LIN {X 0,Y 246.822,Z 659.839,A -85,B 0,C 180,E1 -20933.784,E2 -20933.784} C_VEL
LIN {X 0,Y 240.149,Z 668.993,A -85,B 0,C 180,E1 -20935.712,E2 -20935.712} C_VEL
LIN {X 0,Y 234.092,Z 676.593,A -85,B 0,C 180,E1 -20937.798,E2 -20937.798} C_VEL
LIN {X 0,Y 227.642,Z 683.866,A -85,B 0,C 180,E1 -20940.398,E2 -20940.398} C_VEL
LIN {X 0,Y 222.706,Z 688.862,A -85,B 0,C 180,E1 -20942.769,E2 -20942.769} C_VEL
LIN {X 0,Y 218.214,Z 692.902,A -85,B 0,C 180,E1 -20945.248,E2 -20945.248} C_VEL
LIN {X 0,Y 215.578,Z 695.042,A -85,B 0,C 180,E1 -20946.97,E2 -20946.97} C_VEL
LIN {X 0,Y 211.246,Z 698.163,A -85,B 0,C 180,E1 -20950.568,E2 -20950.568} C_VEL
LIN {X 0,Y 208.028,Z 699.817,A -85,B 0,C 180,E1 -20954.32,E2 -20954.32} C_VEL
LIN {X 0,Y 205.977,Z 699.948,A -85,B 0,C 180,E1 -20958.187,E2 -20958.187} C_VEL
LIN {X 0,Y 204.89,Z 698.61,A -85,B 0,C 180,E1 -20962.114,E2 -20962.114} C_VEL
LIN {X 0,Y 204.811,Z 698.606,A -85,B 0,C 180,E1 -20962.607,E2 -20962.607} C_VEL
LIN {X 0,Y 204.425,Z 700.65,A -85,B 0,C 180,E1 -20966.057,E2 -20966.057} C_VEL
LIN {X 0,Y 204.43,Z 701.266,A -85,B 0,C 180,E1 -20968.03,E2 -20968.03} C_VEL
LIN {X 0,Y 204.516,Z 701.484,A -85,B 0,C 180,E1 -20970,E2 -20970} C_VEL
LIN {X 0,Y 204.399,Z 701.253,A -85,B 0,C 180,E1 -20971.97,E2 -20971.97} C_VEL
LIN {X 0,Y 204.384,Z 700.488,A -85,B 0,C 180,E1 -20974.287,E2 -20974.287} C_VEL
LIN {X 0,Y 204.663,Z 698.173,A -85,B 0,C 180,E1 -20977.895,E2 -20977.895} C_VEL
LIN {X 0,Y 205.307,Z 695.187,A -85,B 0,C 180,E1 -20980.852,E2 -20980.852} C_VEL
LIN {X 0,Y 206.295,Z 691.137,A -85,B 0,C 180,E1 -20983.797,E2 -20983.797} C_VEL
LIN {X 0,Y 208.254,Z 684.908,A -85,B 0,C 180,E1 -20987.175,E2 -20987.175} C_VEL
LIN {X 0,Y 210.401,Z 678.115,A -85,B 0,C 180,E1 -20990.022,E2 -20990.022} C_VEL
LIN {X 0,Y 212.491,Z 671.31,A -85,B 0,C 180,E1 -20992.394,E2 -20992.394} C_VEL
LIN {X 0,Y 217.207,Z 666.561,A -85,B 0,C 180,E1 -20995.901,E2 -20995.901} C_VEL
LIN {X 0,Y 221.61,Z 661.924,A -85,B 0,C 180,E1 -20998.405,E2 -20998.405} C_VEL
LIN {X 0,Y 227.57,Z 655.288,A -85,B 0,C 180,E1 -21001.151,E2 -21001.151} C_VEL
LIN {X 0,Y 234.374,Z 647.105,A -85,B 0,C 180,E1 -21003.693,E2 -21003.693} C_VEL
LIN {X 0,Y 241.865,Z 637.223,A -85,B 0,C 180,E1 -21006.045,E2 -21006.045} C_VEL
LIN {X 0,Y 249.165,Z 626.646,A -85,B 0,C 180,E1 -21007.894,E2 -21007.894} C_VEL
LIN {X 0,Y 255.952,Z 615.572,A -85,B 0,C 180,E1 -21009.418,E2 -21009.418} C_VEL
LIN {X 0,Y 262.663,Z 603.149,A -85,B 0,C 180,E1 -21010.708,E2 -21010.708} C_VEL
LIN {X 0,Y 269.007,Z 589.494,A -85,B 0,C 180,E1 -21011.775,E2 -21011.775} C_VEL
LIN {X 0,Y 275.128,Z 573.285,A -85,B 0,C 180,E1 -21012.729,E2 -21012.729} C_VEL
LIN {X 0,Y 279.953,Z 556.394,A -85,B 0,C 180,E1 -21013.539,E2 -21013.539} C_VEL
LIN {X 0,Y 281.282,Z 550.85,A -85,B 0,C 180,E1 -21013.828,E2 -21013.828} C_VEL
LIN {X 0,Y 282.041,Z 547.448,A -85,B 0,C 180,E1 -21014.196,E2 -21014.196} C_VEL
LIN {X 0,Y 282.381,Z 544.653,A -85,B 0,C 180,E1 -21016.2,E2 -21016.2} C_VEL
LIN {X 0,Y 282.787,Z 543.852,A -85,B 0,C 180,E1 -21017.546,E2 -21017.546} C_VEL
LIN {X 0,Y 277.691,Z 563.088,A -85,B 0,C 180,E1 -21018.619,E2 -21018.619} C_VEL
LIN {X 0,Y 272.938,Z 576.661,A -85,B 0,C 180,E1 -21019.687,E2 -21019.687} C_VEL
LIN {X 0,Y 267.626,Z 588.882,A -85,B 0,C 180,E1 -21020.931,E2 -21020.931} C_VEL
LIN {X 0,Y 261.853,Z 600.028,A -85,B 0,C 180,E1 -21022.367,E2 -21022.367} C_VEL
LIN {X 0,Y 255.179,Z 610.907,A -85,B 0,C 180,E1 -21024.179,E2 -21024.179} C_VEL
LIN {X 0,Y 248.845,Z 619.829,A -85,B 0,C 180,E1 -21026.097,E2 -21026.097} C_VEL
LIN {X 0,Y 242.801,Z 627.197,A -85,B 0,C 180,E1 -21028.112,E2 -21028.112} C_VEL
LIN {X 0,Y 236.398,Z 634.071,A -85,B 0,C 180,E1 -21030.624,E2 -21030.624} C_VEL
LIN {X 0,Y 231.215,Z 638.794,A -85,B 0,C 180,E1 -21032.875,E2 -21032.875} C_VEL
LIN {X 0,Y 225.025,Z 643.457,A -85,B 0,C 180,E1 -21036.045,E2 -21036.045} C_VEL
LIN {X 0,Y 222.181,Z 645.2,A -85,B 0,C 180,E1 -21037.692,E2 -21037.692} C_VEL
LIN {X 0,Y 219.568,Z 646.531,A -85,B 0,C 180,E1 -21039.385,E2 -21039.385} C_VEL
LIN {X 0,Y 217.066,Z 647.461,A -85,B 0,C 180,E1 -21041.109,E2 -21041.109} C_VEL
LIN {X 0,Y 212.867,Z 648.156,A -85,B 0,C 180,E1 -21044.685,E2 -21044.685} C_VEL
LIN {X 0,Y 211.13,Z 647.932,A -85,B 0,C 180,E1 -21046.526,E2 -21046.526} C_VEL
LIN {X 0,Y 208.468,Z 646.274,A -85,B 0,C 180,E1 -21050.296,E2 -21050.296} C_VEL
LIN {X 0,Y 206.567,Z 643.065,A -85,B 0,C 180,E1 -21054.142,E2 -21054.142} C_VEL
LIN {X 0,Y 205.609,Z 639.573,A -85,B 0,C 180,E1 -21057.061,E2 -21057.061} C_VEL
LIN {X 0,Y 205.18,Z 635.056,A -85,B 0,C 180,E1 -21060,E2 -21060} C_VEL
LIN {X 0,Y 205.28,Z 628.361,A -85,B 0,C 180,E1 -21063.435,E2 -21063.435} C_VEL
LIN {X 0,Y 205.557,Z 622.501,A -85,B 0,C 180,E1 -21065.887,E2 -21065.887} C_VEL
LIN {X 0,Y 205.965,Z 613.792,A -85,B 0,C 180,E1 -21068.89,E2 -21068.89} C_VEL
LIN {X 0,Y 206.717,Z 603.469,A -85,B 0,C 180,E1 -21071.77,E2 -21071.77} C_VEL
LIN {X 0,Y 207.701,Z 591.458,A -85,B 0,C 180,E1 -21074.451,E2 -21074.451} C_VEL
LIN {X 0,Y 208.737,Z 579.31,A -85,B 0,C 180,E1 -21076.63,E2 -21076.63} C_VEL
LIN {X 0,Y 209.825,Z 565.811,A -85,B 0,C 180,E1 -21078.554,E2 -21078.554} C_VEL
LIN {X 0,Y 210.638,Z 551.375,A -85,B 0,C 180,E1 -21080.114,E2 -21080.114} C_VEL
LIN {X 0,Y 211.452,Z 537.597,A -85,B 0,C 180,E1 -21081.197,E2 -21081.197} C_VEL
LIN {X 0,Y 214.083,Z 473.822,A -85,B 0,C 180,E1 -21084.869,E2 -21084.869} C_VEL
LIN {X 0,Y 207.846,Z 451.881,A -85,B 0,C 180,E1 -21086.423,E2 -21086.423} C_VEL
LIN {X 0,Y 206.822,Z 447.715,A -85,B 0,C 180,E1 -21086.741,E2 -21086.741} C_VEL
LIN {X 0,Y 206.719,Z 447.71,A -85,B 0,C 180,E1 -21091.794,E2 -21091.794} C_VEL
LIN {X 0,Y 206.701,Z 447.709,A -85,B 0,C 180,E1 -21095.311,E2 -21095.311} C_VEL
LIN {X 0,Y 206.657,Z 447.832,A -85,B 0,C 180,E1 -21099.431,E2 -21099.431} C_VEL
LIN {X 0,Y 207.094,Z 449.45,A -85,B 0,C 180,E1 -21100.15,E2 -21100.15} C_VEL
LIN {X 0,Y 208.097,Z 451.279,A -85,B 0,C 180,E1 -21101.101,E2 -21101.101} C_VEL
LIN {X 0,Y 211.34,Z 459.761,A -85,B 0,C 180,E1 -21104.839,E2 -21104.839} C_VEL
LIN {X 0,Y 214.271,Z 468.248,A -85,B 0,C 180,E1 -21108.223,E2 -21108.223} C_VEL
LIN {X 0,Y 216.652,Z 475.96,A -85,B 0,C 180,E1 -21110.943,E2 -21110.943} C_VEL
LIN {X 0,Y 222.997,Z 488.678,A -85,B 0,C 180,E1 -21112.765,E2 -21112.765} C_VEL
LIN {X 0,Y 228.7,Z 501.914,A -85,B 0,C 180,E1 -21114.352,E2 -21114.352} C_VEL
LIN {X 0,Y 231.099,Z 518.723,A -85,B 0,C 180,E1 -21115.406,E2 -21115.406} C_VEL
LIN {X 0,Y 228.053,Z 586.183,A -85,B 0,C 180,E1 -21117.429,E2 -21117.429} C_VEL
LIN {X 0,Y 226.882,Z 599.328,A -85,B 0,C 180,E1 -21118.093,E2 -21118.093} C_VEL
LIN {X 0,Y 225.302,Z 611.278,A -85,B 0,C 180,E1 -21119.023,E2 -21119.023} C_VEL
LIN {X 0,Y 223.274,Z 622.987,A -85,B 0,C 180,E1 -21120.28,E2 -21120.28} C_VEL
LIN {X 0,Y 220.717,Z 635.03,A -85,B 0,C 180,E1 -21121.987,E2 -21121.987} C_VEL
LIN {X 0,Y 218.056,Z 645.622,A -85,B 0,C 180,E1 -21123.951,E2 -21123.951} C_VEL
LIN {X 0,Y 215.52,Z 654.872,A -85,B 0,C 180,E1 -21126.12,E2 -21126.12} C_VEL
LIN {X 0,Y 212.898,Z 663.681,A -85,B 0,C 180,E1 -21128.708,E2 -21128.708} C_VEL
LIN {X 0,Y 210.376,Z 671.148,A -85,B 0,C 180,E1 -21131.496,E2 -21131.496} C_VEL
LIN {X 0,Y 208.434,Z 677.133,A -85,B 0,C 180,E1 -21134.351,E2 -21134.351} C_VEL
LIN {X 0,Y 206.83,Z 681.865,A -85,B 0,C 180,E1 -21137.24,E2 -21137.24} C_VEL
LIN {X 0,Y 205.714,Z 685.481,A -85,B 0,C 180,E1 -21140.164,E2 -21140.164} C_VEL
LIN {X 0,Y 205.197,Z 687.34,A -85,B 0,C 180,E1 -21142.126,E2 -21142.126} C_VEL
LIN {X 0,Y 204.763,Z 688.973,A -85,B 0,C 180,E1 -21144.479,E2 -21144.479} C_VEL
LIN {X 0,Y 204.472,Z 690.36,A -85,B 0,C 180,E1 -21148.03,E2 -21148.03} C_VEL
LIN {X 0,Y 204.474,Z 690.59,A -85,B 0,C 180,E1 -21150,E2 -21150} C_VEL
LIN {X 0,Y 204.471,Z 690.394,A -85,B 0,C 180,E1 -21151.97,E2 -21151.97} C_VEL
LIN {X 0,Y 204.823,Z 688.834,A -85,B 0,C 180,E1 -21155.908,E2 -21155.908} C_VEL
LIN {X 0,Y 205.193,Z 687.462,A -85,B 0,C 180,E1 -21157.874,E2 -21157.874} C_VEL
LIN {X 0,Y 206.024,Z 684.579,A -85,B 0,C 180,E1 -21160.814,E2 -21160.814} C_VEL
LIN {X 0,Y 207.272,Z 680.658,A -85,B 0,C 180,E1 -21163.73,E2 -21163.73} C_VEL
LIN {X 0,Y 208.976,Z 675.573,A -85,B 0,C 180,E1 -21166.61,E2 -21166.61} C_VEL
LIN {X 0,Y 211.126,Z 669.161,A -85,B 0,C 180,E1 -21169.444,E2 -21169.444} C_VEL
LIN {X 0,Y 213.778,Z 661.188,A -85,B 0,C 180,E1 -21172.214,E2 -21172.214} C_VEL
LIN {X 0,Y 216.312,Z 652.44,A -85,B 0,C 180,E1 -21174.642,E2 -21174.642} C_VEL
LIN {X 0,Y 218.833,Z 642.979,A -85,B 0,C 180,E1 -21176.719,E2 -21176.719} C_VEL
LIN {X 0,Y 221.597,Z 631.665,A -85,B 0,C 180,E1 -21178.665,E2 -21178.665} C_VEL
LIN {X 0,Y 223.833,Z 620.502,A -85,B 0,C 180,E1 -21180.157,E2 -21180.157} C_VEL
LIN {X 0,Y 225.952,Z 607.822,A -85,B 0,C 180,E1 -21181.399,E2 -21181.399} C_VEL
LIN {X 0,Y 227.283,Z 596.137,A -85,B 0,C 180,E1 -21182.236,E2 -21182.236} C_VEL
LIN {X 0,Y 228.293,Z 583.8,A -85,B 0,C 180,E1 -21182.794,E2 -21182.794} C_VEL
LIN {X 0,Y 231.175,Z 518.266,A -85,B 0,C 180,E1 -21184.746,E2 -21184.746} C_VEL
LIN {X 0,Y 228.56,Z 501.373,A -85,B 0,C 180,E1 -21185.844,E2 -21185.844} C_VEL
LIN {X 0,Y 222.629,Z 487.777,A -85,B 0,C 180,E1 -21187.498,E2 -21187.498} C_VEL
LIN {X 0,Y 216.547,Z 475.617,A -85,B 0,C 180,E1 -21189.3,E2 -21189.3} C_VEL
LIN {X 0,Y 213.479,Z 465.768,A -85,B 0,C 180,E1 -21192.903,E2 -21192.903} C_VEL
LIN {X 0,Y 210.639,Z 457.862,A -85,B 0,C 180,E1 -21196.186,E2 -21196.186} C_VEL
LIN {X 0,Y 207.768,Z 450.735,A -85,B 0,C 180,E1 -21199.388,E2 -21199.388} C_VEL
LIN {X 0,Y 206.681,Z 447.744,A -85,B 0,C 180,E1 -21200.807,E2 -21200.807} C_VEL
LIN {X 0,Y 206.798,Z 447.743,A -85,B 0,C 180,E1 -21204.357,E2 -21204.357} C_VEL
LIN {X 0,Y 210.172,Z 463.929,A -85,B 0,C 180,E1 -21209.061,E2 -21209.061} C_VEL
LIN {X 0,Y 212.003,Z 472.76,A -85,B 0,C 180,E1 -21211.54,E2 -21211.54} C_VEL
LIN {X 0,Y 211.794,Z 476.671,A -85,B 0,C 180,E1 -21212.515,E2 -21212.515} C_VEL
LIN {X 0,Y 213.201,Z 497.323,A -85,B 0,C 180,E1 -21213.773,E2 -21213.773} C_VEL
LIN {X 0,Y 214.619,Z 511.272,A -85,B 0,C 180,E1 -21214.629,E2 -21214.629} C_VEL
LIN {X 0,Y 210.995,Z 588.15,A -85,B 0,C 180,E1 -21219.055,E2 -21219.055} C_VEL
LIN {X 0,Y 210.145,Z 602.588,A -85,B 0,C 180,E1 -21220.272,E2 -21220.272} C_VEL
LIN {X 0,Y 209.238,Z 614.678,A -85,B 0,C 180,E1 -21221.646,E2 -21221.646} C_VEL
LIN {X 0,Y 208.238,Z 627.949,A -85,B 0,C 180,E1 -21223.581,E2 -21223.581} C_VEL
LIN {X 0,Y 207.079,Z 640.895,A -85,B 0,C 180,E1 -21226.006,E2 -21226.006} C_VEL
LIN {X 0,Y 206.541,Z 646.882,A -85,B 0,C 180,E1 -21227.351,E2 -21227.351} C_VEL
LIN {X 0,Y 205.425,Z 651.21,A -85,B 0,C 180,E1 -21228.448,E2 -21228.448} C_VEL
LIN {X 0,Y 202.035,Z 657.624,A -85,B 0,C 180,E1 -21230.368,E2 -21230.368} C_VEL
LIN {X 0,Y 198.845,Z 663.489,A -85,B 0,C 180,E1 -21232.472,E2 -21232.472} C_VEL
LIN {X 0,Y 198.045,Z 667.005,A -85,B 0,C 180,E1 -21233.822,E2 -21233.822} C_VEL
LIN {X 0,Y 197.791,Z 674.226,A -85,B 0,C 180,E1 -21236.945,E2 -21236.945} C_VEL
LIN {X 0,Y 197.636,Z 679.846,A -85,B 0,C 180,E1 -21240,E2 -21240} C_VEL
LIN {X 0,Y 197.667,Z 684.221,A -85,B 0,C 180,E1 -21243.057,E2 -21243.057} C_VEL
LIN {X 0,Y 197.997,Z 687.774,A -85,B 0,C 180,E1 -21246.342,E2 -21246.342} C_VEL
LIN {X 0,Y 199.157,Z 690.616,A -85,B 0,C 180,E1 -21250.163,E2 -21250.163} C_VEL
LIN {X 0,Y 200.099,Z 691.561,A -85,B 0,C 180,E1 -21252.165,E2 -21252.165} C_VEL
LIN {X 0,Y 202.85,Z 692.291,A -85,B 0,C 180,E1 -21256.091,E2 -21256.091} C_VEL
LIN {X 0,Y 206.515,Z 691.591,A -85,B 0,C 180,E1 -21259.896,E2 -21259.896} C_VEL
LIN {X 0,Y 211.509,Z 689.338,A -85,B 0,C 180,E1 -21263.499,E2 -21263.499} C_VEL
LIN {X 0,Y 217.38,Z 685.573,A -85,B 0,C 180,E1 -21266.912,E2 -21266.912} C_VEL
LIN {X 0,Y 222.428,Z 681.658,A -85,B 0,C 180,E1 -21269.324,E2 -21269.324} C_VEL
LIN {X 0,Y 227.95,Z 676.712,A -85,B 0,C 180,E1 -21271.61,E2 -21271.61} C_VEL
LIN {X 0,Y 234.961,Z 669.564,A -85,B 0,C 180,E1 -21274.114,E2 -21274.114} C_VEL
LIN {X 0,Y 242.537,Z 660.638,A -85,B 0,C 180,E1 -21276.443,E2 -21276.443} C_VEL
LIN {X 0,Y 249.499,Z 651.211,A -85,B 0,C 180,E1 -21278.295,E2 -21278.295} C_VEL
LIN {X 0,Y 256.842,Z 639.775,A -85,B 0,C 180,E1 -21280.019,E2 -21280.019} C_VEL
LIN {X 0,Y 263.232,Z 628.029,A -85,B 0,C 180,E1 -21281.361,E2 -21281.361} C_VEL
LIN {X 0,Y 269.285,Z 614.812,A -85,B 0,C 180,E1 -21282.478,E2 -21282.478} C_VEL
LIN {X 0,Y 273.318,Z 604.09,A -85,B 0,C 180,E1 -21283.161,E2 -21283.161} C_VEL
LIN {X 0,Y 277.995,Z 588.116,A -85,B 0,C 180,E1 -21283.92,E2 -21283.92} C_VEL
LIN {X 0,Y 283.776,Z 566.322,A -85,B 0,C 180,E1 -21284.857,E2 -21284.857} C_VEL
LIN {X 0,Y 283.782,Z 566.28,A -85,B 0,C 180,E1 -21284.988,E2 -21284.988} C_VEL
LIN {X 0,Y 274.469,Z 600.667,A -85,B 0,C 180,E1 -21286.489,E2 -21286.489} C_VEL
LIN {X 0,Y 269.264,Z 615.152,A -85,B 0,C 180,E1 -21287.264,E2 -21287.264} C_VEL
LIN {X 0,Y 263.479,Z 628.141,A -85,B 0,C 180,E1 -21288.176,E2 -21288.176} C_VEL
LIN {X 0,Y 257.251,Z 639.905,A -85,B 0,C 180,E1 -21289.288,E2 -21289.288} C_VEL
LIN {X 0,Y 251.316,Z 649.663,A -85,B 0,C 180,E1 -21290.491,E2 -21290.491} C_VEL
LIN {X 0,Y 243.861,Z 660.474,A -85,B 0,C 180,E1 -21292.235,E2 -21292.235} C_VEL
LIN {X 0,Y 236.866,Z 669.428,A -85,B 0,C 180,E1 -21294.126,E2 -21294.126} C_VEL
LIN {X 0,Y 230.383,Z 676.825,A -85,B 0,C 180,E1 -21296.17,E2 -21296.17} C_VEL
LIN {X 0,Y 223.515,Z 683.927,A -85,B 0,C 180,E1 -21298.747,E2 -21298.747} C_VEL
LIN {X 0,Y 216.518,Z 690.243,A -85,B 0,C 180,E1 -21301.923,E2 -21301.923} C_VEL
LIN {X 0,Y 211.85,Z 693.85,A -85,B 0,C 180,E1 -21304.452,E2 -21304.452} C_VEL
LIN {X 0,Y 209.116,Z 695.783,A -85,B 0,C 180,E1 -21306.215,E2 -21306.215} C_VEL
LIN {X 0,Y 204.568,Z 698.452,A -85,B 0,C 180,E1 -21309.906,E2 -21309.906} C_VEL
LIN {X 0,Y 201.182,Z 699.686,A -85,B 0,C 180,E1 -21313.771,E2 -21313.771} C_VEL
LIN {X 0,Y 199.019,Z 699.489,A -85,B 0,C 180,E1 -21317.767,E2 -21317.767} C_VEL
LIN {X 0,Y 197.914,Z 697.929,A -85,B 0,C 180,E1 -21321.705,E2 -21321.705} C_VEL
LIN {X 0,Y 197.348,Z 700.363,A -85,B 0,C 180,E1 -21325.668,E2 -21325.668} C_VEL
LIN {X 0,Y 197.334,Z 701.077,A -85,B 0,C 180,E1 -21327.959,E2 -21327.959} C_VEL
LIN {X 0,Y 197.414,Z 701.295,A -85,B 0,C 180,E1 -21330,E2 -21330} C_VEL
LIN {X 0,Y 197.303,Z 701.064,A -85,B 0,C 180,E1 -21332.041,E2 -21332.041} C_VEL
LIN {X 0,Y 197.286,Z 700.44,A -85,B 0,C 180,E1 -21334.086,E2 -21334.086} C_VEL
LIN {X 0,Y 197.366,Z 699.423,A -85,B 0,C 180,E1 -21336.132,E2 -21336.132} C_VEL
LIN {X 0,Y 197.608,Z 697.982,A -85,B 0,C 180,E1 -21338.179,E2 -21338.179} C_VEL
LIN {X 0,Y 198.292,Z 694.996,A -85,B 0,C 180,E1 -21341.241,E2 -21341.241} C_VEL
LIN {X 0,Y 199.367,Z 690.947,A -85,B 0,C 180,E1 -21344.286,E2 -21344.286} C_VEL
LIN {X 0,Y 201.469,Z 684.719,A -85,B 0,C 180,E1 -21347.772,E2 -21347.772} C_VEL
LIN {X 0,Y 203.708,Z 678,A -85,B 0,C 180,E1 -21350.678,E2 -21350.678} C_VEL
LIN {X 0,Y 205.782,Z 671.436,A -85,B 0,C 180,E1 -21353.02,E2 -21353.02} C_VEL
LIN {X 0,Y 209.471,Z 668.21,A -85,B 0,C 180,E1 -21355.86,E2 -21355.86} C_VEL
LIN {X 0,Y 215.452,Z 662.758,A -85,B 0,C 180,E1 -21359.295,E2 -21359.295} C_VEL
LIN {X 0,Y 220.662,Z 657.61,A -85,B 0,C 180,E1 -21361.703,E2 -21361.703} C_VEL
LIN {X 0,Y 227.571,Z 650.286,A -85,B 0,C 180,E1 -21364.306,E2 -21364.306} C_VEL
LIN {X 0,Y 235.199,Z 641.371,A -85,B 0,C 180,E1 -21366.7,E2 -21366.7} C_VEL
LIN {X 0,Y 242.388,Z 632.189,A -85,B 0,C 180,E1 -21368.565,E2 -21368.565} C_VEL
LIN {X 0,Y 250.724,Z 620.207,A -85,B 0,C 180,E1 -21370.407,E2 -21370.407} C_VEL
LIN {X 0,Y 257.612,Z 609.046,A -85,B 0,C 180,E1 -21371.681,E2 -21371.681} C_VEL
LIN {X 0,Y 264.024,Z 597.055,A -85,B 0,C 180,E1 -21372.749,E2 -21372.749} C_VEL
LIN {X 0,Y 270.001,Z 584.082,A -85,B 0,C 180,E1 -21373.613,E2 -21373.613} C_VEL
LIN {X 0,Y 275.91,Z 568.177,A -85,B 0,C 180,E1 -21374.473,E2 -21374.473} C_VEL
LIN {X 0,Y 280.208,Z 553.135,A -85,B 0,C 180,E1 -21375.19,E2 -21375.19} C_VEL
LIN {X 0,Y 280.581,Z 551.39,A -85,B 0,C 180,E1 -21376.459,E2 -21376.459} C_VEL
LIN {X 0,Y 276.191,Z 566.287,A -85,B 0,C 180,E1 -21377.311,E2 -21377.311} C_VEL
LIN {X 0,Y 271.097,Z 579.588,A -85,B 0,C 180,E1 -21378.37,E2 -21378.37} C_VEL
LIN {X 0,Y 265.538,Z 591.332,A -85,B 0,C 180,E1 -21379.576,E2 -21379.576} C_VEL
LIN {X 0,Y 259.479,Z 602.124,A -85,B 0,C 180,E1 -21380.97,E2 -21380.97} C_VEL
LIN {X 0,Y 252.485,Z 612.737,A -85,B 0,C 180,E1 -21382.741,E2 -21382.741} C_VEL
LIN {X 0,Y 245.778,Z 621.454,A -85,B 0,C 180,E1 -21384.616,E2 -21384.616} C_VEL
LIN {X 0,Y 239.425,Z 628.646,A -85,B 0,C 180,E1 -21386.607,E2 -21386.607} C_VEL
LIN {X 0,Y 232.565,Z 635.41,A -85,B 0,C 180,E1 -21389.087,E2 -21389.087} C_VEL
LIN {X 0,Y 227.034,Z 640.032,A -85,B 0,C 180,E1 -21391.327,E2 -21391.327} C_VEL
LIN {X 0,Y 221.97,Z 643.629,A -85,B 0,C 180,E1 -21393.688,E2 -21393.688} C_VEL
LIN {X 0,Y 215.84,Z 646.984,A -85,B 0,C 180,E1 -21397,E2 -21397} C_VEL
LIN {X 0,Y 210.484,Z 648.819,A -85,B 0,C 180,E1 -21400.494,E2 -21400.494} C_VEL
LIN {X 0,Y 208.172,Z 649.157,A -85,B 0,C 180,E1 -21402.311,E2 -21402.311} C_VEL
LIN {X 0,Y 204.295,Z 648.646,A -85,B 0,C 180,E1 -21406.066,E2 -21406.066} C_VEL
LIN {X 0,Y 201.482,Z 646.632,A -85,B 0,C 180,E1 -21409.956,E2 -21409.956} C_VEL
LIN {X 0,Y 199.926,Z 644.09,A -85,B 0,C 180,E1 -21412.933,E2 -21412.933} C_VEL
LIN {X 0,Y 198.796,Z 640.612,A -85,B 0,C 180,E1 -21415.946,E2 -21415.946} C_VEL
LIN {X 0,Y 198.185,Z 636.15,A -85,B 0,C 180,E1 -21418.984,E2 -21418.984} C_VEL
LIN {X 0,Y 198.127,Z 629.595,A -85,B 0,C 180,E1 -21422.541,E2 -21422.541} C_VEL
LIN {X 0,Y 198.487,Z 622.498,A -85,B 0,C 180,E1 -21425.588,E2 -21425.588} C_VEL
LIN {X 0,Y 198.945,Z 612.604,A -85,B 0,C 180,E1 -21429.014,E2 -21429.014} C_VEL
LIN {X 0,Y 199.625,Z 603.128,A -85,B 0,C 180,E1 -21431.68,E2 -21431.68} C_VEL
LIN {X 0,Y 200.532,Z 592.251,A -85,B 0,C 180,E1 -21434.201,E2 -21434.201} C_VEL
LIN {X 0,Y 201.579,Z 580.137,A -85,B 0,C 180,E1 -21436.456,E2 -21436.456} C_VEL
LIN {X 0,Y 202.683,Z 566.679,A -85,B 0,C 180,E1 -21438.446,E2 -21438.446} C_VEL
LIN {X 0,Y 203.5,Z 552.191,A -85,B 0,C 180,E1 -21440.072,E2 -21440.072} C_VEL
LIN {X 0,Y 204.348,Z 538.166,A -85,B 0,C 180,E1 -21441.215,E2 -21441.215} C_VEL
LIN {X 0,Y 207.015,Z 475.033,A -85,B 0,C 180,E1 -21445.05,E2 -21445.05} C_VEL
LIN {X 0,Y 200.002,Z 449.697,A -85,B 0,C 180,E1 -21446.869,E2 -21446.869} C_VEL
LIN {X 0,Y 199.767,Z 448.592,A -85,B 0,C 180,E1 -21447.019,E2 -21447.019} C_VEL
LIN {X 0,Y 199.673,Z 448.58,A -85,B 0,C 180,E1 -21452.355,E2 -21452.355} C_VEL
LIN {X 0,Y 199.64,Z 448.761,A -85,B 0,C 180,E1 -21457.392,E2 -21457.392} C_VEL
LIN {X 0,Y 203.405,Z 457.918,A -85,B 0,C 180,E1 -21461.939,E2 -21461.939} C_VEL
LIN {X 0,Y 206.501,Z 466.346,A -85,B 0,C 180,E1 -21465.62,E2 -21465.62} C_VEL
LIN {X 0,Y 209.628,Z 475.979,A -85,B 0,C 180,E1 -21469.363,E2 -21469.363} C_VEL
LIN {X 0,Y 216.333,Z 488.945,A -85,B 0,C 180,E1 -21471.418,E2 -21471.418} C_VEL
LIN {X 0,Y 222.514,Z 502.914,A -85,B 0,C 180,E1 -21473.237,E2 -21473.237} C_VEL
LIN {X 0,Y 223.279,Z 505.55,A -85,B 0,C 180,E1 -21473.488,E2 -21473.488} C_VEL
LIN {X 0,Y 225.25,Z 520.075,A -85,B 0,C 180,E1 -21474.421,E2 -21474.421} C_VEL
LIN {X 0,Y 222.207,Z 584.978,A -85,B 0,C 180,E1 -21476.393,E2 -21476.393} C_VEL
LIN {X 0,Y 221.003,Z 598.633,A -85,B 0,C 180,E1 -21477.071,E2 -21477.071} C_VEL
LIN {X 0,Y 219.423,Z 610.305,A -85,B 0,C 180,E1 -21477.961,E2 -21477.961} C_VEL
LIN {X 0,Y 217.513,Z 621.46,A -85,B 0,C 180,E1 -21479.14,E2 -21479.14} C_VEL
LIN {X 0,Y 215.13,Z 632.451,A -85,B 0,C 180,E1 -21480.657,E2 -21480.657} C_VEL
LIN {X 0,Y 212.278,Z 643.655,A -85,B 0,C 180,E1 -21482.654,E2 -21482.654} C_VEL
LIN {X 0,Y 209.499,Z 653.539,A -85,B 0,C 180,E1 -21484.927,E2 -21484.927} C_VEL
LIN {X 0,Y 206.817,Z 662.418,A -85,B 0,C 180,E1 -21487.524,E2 -21487.524} C_VEL
LIN {X 0,Y 204.032,Z 670.221,A -85,B 0,C 180,E1 -21490.376,E2 -21490.376} C_VEL
LIN {X 0,Y 202.205,Z 675.485,A -85,B 0,C 180,E1 -21492.816,E2 -21492.816} C_VEL
LIN {X 0,Y 200.421,Z 680.625,A -85,B 0,C 180,E1 -21495.791,E2 -21495.791} C_VEL
LIN {X 0,Y 199.056,Z 684.602,A -85,B 0,C 180,E1 -21498.803,E2 -21498.803} C_VEL
LIN {X 0,Y 198.16,Z 687.53,A -85,B 0,C 180,E1 -21501.844,E2 -21501.844} C_VEL
LIN {X 0,Y 197.64,Z 689.372,A -85,B 0,C 180,E1 -21504.669,E2 -21504.669} C_VEL
LIN {X 0,Y 197.38,Z 690.55,A -85,B 0,C 180,E1 -21507.959,E2 -21507.959} C_VEL
LIN {X 0,Y 197.377,Z 690.779,A -85,B 0,C 180,E1 -21510,E2 -21510} C_VEL
LIN {X 0,Y 197.379,Z 690.583,A -85,B 0,C 180,E1 -21512.041,E2 -21512.041} C_VEL
LIN {X 0,Y 197.765,Z 689.023,A -85,B 0,C 180,E1 -21516.12,E2 -21516.12} C_VEL
LIN {X 0,Y 198.156,Z 687.65,A -85,B 0,C 180,E1 -21518.156,E2 -21518.156} C_VEL
LIN {X 0,Y 199.043,Z 684.767,A -85,B 0,C 180,E1 -21521.198,E2 -21521.198} C_VEL
LIN {X 0,Y 200.375,Z 680.845,A -85,B 0,C 180,E1 -21524.213,E2 -21524.213} C_VEL
LIN {X 0,Y 202.171,Z 675.759,A -85,B 0,C 180,E1 -21527.187,E2 -21527.187} C_VEL
LIN {X 0,Y 204.44,Z 669.345,A -85,B 0,C 180,E1 -21530.107,E2 -21530.107} C_VEL
LIN {X 0,Y 207.217,Z 661.37,A -85,B 0,C 180,E1 -21532.957,E2 -21532.957} C_VEL
LIN {X 0,Y 209.769,Z 652.942,A -85,B 0,C 180,E1 -21535.37,E2 -21535.37} C_VEL
LIN {X 0,Y 212.197,Z 644.293,A -85,B 0,C 180,E1 -21537.358,E2 -21537.358} C_VEL
LIN {X 0,Y 215.093,Z 633.217,A -85,B 0,C 180,E1 -21539.348,E2 -21539.348} C_VEL
LIN {X 0,Y 217.394,Z 622.409,A -85,B 0,C 180,E1 -21540.878,E2 -21540.878} C_VEL
LIN {X 0,Y 219.596,Z 610.438,A -85,B 0,C 180,E1 -21542.146,E2 -21542.146} C_VEL
LIN {X 0,Y 221.223,Z 597.119,A -85,B 0,C 180,E1 -21543.163,E2 -21543.163} C_VEL
LIN {X 0,Y 222.368,Z 583.874,A -85,B 0,C 180,E1 -21543.784,E2 -21543.784} C_VEL
LIN {X 0,Y 225.338,Z 519.158,A -85,B 0,C 180,E1 -21545.749,E2 -21545.749} C_VEL
LIN {X 0,Y 223.066,Z 504.133,A -85,B 0,C 180,E1 -21546.762,E2 -21546.762} C_VEL
LIN {X 0,Y 217.296,Z 490.844,A -85,B 0,C 180,E1 -21548.459,E2 -21548.459} C_VEL
LIN {X 0,Y 210.809,Z 478.231,A -85,B 0,C 180,E1 -21550.428,E2 -21550.428} C_VEL
LIN {X 0,Y 209.647,Z 475.903,A -85,B 0,C 180,E1 -21550.811,E2 -21550.811} C_VEL
LIN {X 0,Y 206.653,Z 466.675,A -85,B 0,C 180,E1 -21554.423,E2 -21554.423} C_VEL
LIN {X 0,Y 203.605,Z 458.398,A -85,B 0,C 180,E1 -21558.042,E2 -21558.042} C_VEL
LIN {X 0,Y 201.137,Z 452.241,A -85,B 0,C 180,E1 -21561.027,E2 -21561.027} C_VEL
LIN {X 0,Y 199.749,Z 449.144,A -85,B 0,C 180,E1 -21562.632,E2 -21562.632} C_VEL
LIN {X 0,Y 199.673,Z 448.59,A -85,B 0,C 180,E1 -21562.932,E2 -21562.932} C_VEL
LIN {X 0,Y 199.762,Z 448.686,A -85,B 0,C 180,E1 -21564.068,E2 -21564.068} C_VEL
LIN {X 0,Y 203.011,Z 464.297,A -85,B 0,C 180,E1 -21568.716,E2 -21568.716} C_VEL
LIN {X 0,Y 204.886,Z 473.271,A -85,B 0,C 180,E1 -21571.299,E2 -21571.299} C_VEL
LIN {X 0,Y 204.812,Z 476.502,A -85,B 0,C 180,E1 -21572.183,E2 -21572.183} C_VEL
LIN {X 0,Y 205.979,Z 495.317,A -85,B 0,C 180,E1 -21573.366,E2 -21573.366} C_VEL
LIN {X 0,Y 207.574,Z 511.941,A -85,B 0,C 180,E1 -21574.425,E2 -21574.425} C_VEL
LIN {X 0,Y 203.933,Z 587.529,A -85,B 0,C 180,E1 -21579.01,E2 -21579.01} C_VEL
LIN {X 0,Y 203.061,Z 602.23,A -85,B 0,C 180,E1 -21580.278,E2 -21580.278} C_VEL
LIN {X 0,Y 202.101,Z 614.893,A -85,B 0,C 180,E1 -21581.761,E2 -21581.761} C_VEL
LIN {X 0,Y 201.11,Z 628.159,A -85,B 0,C 180,E1 -21583.765,E2 -21583.765} C_VEL
LIN {X 0,Y 199.951,Z 641.099,A -85,B 0,C 180,E1 -21586.275,E2 -21586.275} C_VEL
LIN {X 0,Y 199.085,Z 651.512,A -85,B 0,C 180,E1 -21588.804,E2 -21588.804} C_VEL
LIN {X 0,Y 198.474,Z 660.051,A -85,B 0,C 180,E1 -21591.344,E2 -21591.344} C_VEL
LIN {X 0,Y 198.045,Z 667.005,A -85,B 0,C 180,E1 -21593.822,E2 -21593.822} C_VEL
LIN {X 0,Y 197.253,Z 670.353,A -85,B 0,C 180,E1 -21595.212,E2 -21595.212} C_VEL
LIN {X 0,Y 195.562,Z 673.25,A -85,B 0,C 180,E1 -21596.645,E2 -21596.645} C_VEL
LIN {X 0,Y 191.279,Z 679.034,A -85,B 0,C 180,E1 -21600.213,E2 -21600.213} C_VEL
LIN {X 0,Y 190.64,Z 681.414,A -85,B 0,C 180,E1 -21601.846,E2 -21601.846} C_VEL
LIN {X 0,Y 190.755,Z 685.417,A -85,B 0,C 180,E1 -21604.955,E2 -21604.955} C_VEL
LIN {X 0,Y 191.471,Z 688.782,A -85,B 0,C 180,E1 -21608.443,E2 -21608.443} C_VEL
LIN {X 0,Y 193.176,Z 691.387,A -85,B 0,C 180,E1 -21612.608,E2 -21612.608} C_VEL
LIN {X 0,Y 196.043,Z 692.543,A -85,B 0,C 180,E1 -21616.666,E2 -21616.666} C_VEL
LIN {X 0,Y 199.904,Z 692.233,A -85,B 0,C 180,E1 -21620.583,E2 -21620.583} C_VEL
LIN {X 0,Y 205.122,Z 690.44,A -85,B 0,C 180,E1 -21624.277,E2 -21624.277} C_VEL
LIN {X 0,Y 211.232,Z 687.19,A -85,B 0,C 180,E1 -21627.762,E2 -21627.762} C_VEL
LIN {X 0,Y 216.487,Z 683.675,A -85,B 0,C 180,E1 -21630.211,E2 -21630.211} C_VEL
LIN {X 0,Y 224.234,Z 677.491,A -85,B 0,C 180,E1 -21633.264,E2 -21633.264} C_VEL
LIN {X 0,Y 231.676,Z 670.514,A -85,B 0,C 180,E1 -21635.729,E2 -21635.729} C_VEL
LIN {X 0,Y 238.488,Z 663.171,A -85,B 0,C 180,E1 -21637.697,E2 -21637.697} C_VEL
LIN {X 0,Y 245.903,Z 654.136,A -85,B 0,C 180,E1 -21639.554,E2 -21639.554} C_VEL
LIN {X 0,Y 253.34,Z 643.548,A -85,B 0,C 180,E1 -21641.213,E2 -21641.213} C_VEL
LIN {X 0,Y 260.606,Z 631.62,A -85,B 0,C 180,E1 -21642.634,E2 -21642.634} C_VEL
LIN {X 0,Y 266.883,Z 619.163,A -85,B 0,C 180,E1 -21643.73,E2 -21643.73} C_VEL
LIN {X 0,Y 271.883,Z 607.224,A -85,B 0,C 180,E1 -21644.521,E2 -21644.521} C_VEL
LIN {X 0,Y 273.263,Z 603.439,A -85,B 0,C 180,E1 -21644.716,E2 -21644.716} C_VEL
LIN {X 0,Y 273.614,Z 602.397,A -85,B 0,C 180,E1 -21645.06,E2 -21645.06} C_VEL
LIN {X 0,Y 267.529,Z 617.887,A -85,B 0,C 180,E1 -21645.88,E2 -21645.88} C_VEL
LIN {X 0,Y 262.535,Z 628.374,A -85,B 0,C 180,E1 -21646.601,E2 -21646.601} C_VEL
LIN {X 0,Y 256.585,Z 638.995,A -85,B 0,C 180,E1 -21647.558,E2 -21647.558} C_VEL
LIN {X 0,Y 250.258,Z 648.943,A -85,B 0,C 180,E1 -21648.704,E2 -21648.704} C_VEL
LIN {X 0,Y 242.411,Z 659.701,A -85,B 0,C 180,E1 -21650.37,E2 -21650.37} C_VEL
LIN {X 0,Y 234.961,Z 668.678,A -85,B 0,C 180,E1 -21652.18,E2 -21652.18} C_VEL
LIN {X 0,Y 226.92,Z 677.253,A -85,B 0,C 180,E1 -21654.499,E2 -21654.499} C_VEL
LIN {X 0,Y 219.589,Z 684.08,A -85,B 0,C 180,E1 -21657.037,E2 -21657.037} C_VEL
LIN {X 0,Y 213.892,Z 688.868,A -85,B 0,C 180,E1 -21659.383,E2 -21659.383} C_VEL
LIN {X 0,Y 207.094,Z 693.766,A -85,B 0,C 180,E1 -21662.733,E2 -21662.733} C_VEL
LIN {X 0,Y 202.672,Z 696.405,A -85,B 0,C 180,E1 -21665.41,E2 -21665.41} C_VEL
LIN {X 0,Y 197.924,Z 698.669,A -85,B 0,C 180,E1 -21669.201,E2 -21669.201} C_VEL
LIN {X 0,Y 194.358,Z 699.47,A -85,B 0,C 180,E1 -21673.185,E2 -21673.185} C_VEL
LIN {X 0,Y 192.097,Z 698.87,A -85,B 0,C 180,E1 -21677.319,E2 -21677.319} C_VEL
LIN {X 0,Y 190.993,Z 697.401,A -85,B 0,C 180,E1 -21681.003,E2 -21681.003} C_VEL
LIN {X 0,Y 190.436,Z 699.266,A -85,B 0,C 180,E1 -21683.643,E2 -21683.643} C_VEL
LIN {X 0,Y 190.241,Z 700.888,A -85,B 0,C 180,E1 -21687.883,E2 -21687.883} C_VEL
LIN {X 0,Y 190.315,Z 701.106,A -85,B 0,C 180,E1 -21690,E2 -21690} C_VEL
LIN {X 0,Y 190.189,Z 700.393,A -85,B 0,C 180,E1 -21693.864,E2 -21693.864} C_VEL
LIN {X 0,Y 190.296,Z 699.234,A -85,B 0,C 180,E1 -21696.361,E2 -21696.361} C_VEL
LIN {X 0,Y 190.554,Z 697.792,A -85,B 0,C 180,E1 -21698.484,E2 -21698.484} C_VEL
LIN {X 0,Y 191.298,Z 694.806,A -85,B 0,C 180,E1 -21701.658,E2 -21701.658} C_VEL
LIN {X 0,Y 192.454,Z 690.757,A -85,B 0,C 180,E1 -21704.811,E2 -21704.811} C_VEL
LIN {X 0,Y 194.7,Z 684.53,A -85,B 0,C 180,E1 -21708.412,E2 -21708.412} C_VEL
LIN {X 0,Y 197.048,Z 677.819,A -85,B 0,C 180,E1 -21711.407,E2 -21711.407} C_VEL
LIN {X 0,Y 199.216,Z 671.316,A -85,B 0,C 180,E1 -21713.797,E2 -21713.797} C_VEL
LIN {X 0,Y 204.58,Z 667.331,A -85,B 0,C 180,E1 -21717.631,E2 -21717.631} C_VEL
LIN {X 0,Y 209.325,Z 663.483,A -85,B 0,C 180,E1 -21720.24,E2 -21720.24} C_VEL
LIN {X 0,Y 216.694,Z 656.985,A -85,B 0,C 180,E1 -21723.46,E2 -21723.46} C_VEL
LIN {X 0,Y 224.047,Z 649.877,A -85,B 0,C 180,E1 -21726.027,E2 -21726.027} C_VEL
LIN {X 0,Y 232.053,Z 641.234,A -85,B 0,C 180,E1 -21728.38,E2 -21728.38} C_VEL
LIN {X 0,Y 240.596,Z 631.096,A -85,B 0,C 180,E1 -21730.393,E2 -21730.393} C_VEL
LIN {X 0,Y 248.987,Z 619.745,A -85,B 0,C 180,E1 -21732.096,E2 -21732.096} C_VEL
LIN {X 0,Y 256.897,Z 607.612,A -85,B 0,C 180,E1 -21733.421,E2 -21733.421} C_VEL
LIN {X 0,Y 263.598,Z 595.662,A -85,B 0,C 180,E1 -21734.417,E2 -21734.417} C_VEL
LIN {X 0,Y 270.901,Z 580.153,A -85,B 0,C 180,E1 -21735.363,E2 -21735.363} C_VEL
LIN {X 0,Y 274.376,Z 571.335,A -85,B 0,C 180,E1 -21735.825,E2 -21735.825} C_VEL
LIN {X 0,Y 274.045,Z 572.065,A -85,B 0,C 180,E1 -21736.177,E2 -21736.177} C_VEL
LIN {X 0,Y 268.818,Z 584.094,A -85,B 0,C 180,E1 -21737.176,E2 -21737.176} C_VEL
LIN {X 0,Y 263.009,Z 595.162,A -85,B 0,C 180,E1 -21738.341,E2 -21738.341} C_VEL
LIN {X 0,Y 256.091,Z 606.307,A -85,B 0,C 180,E1 -21739.84,E2 -21739.84} C_VEL
LIN {X 0,Y 248.78,Z 616.275,A -85,B 0,C 180,E1 -21741.574,E2 -21741.574} C_VEL
LIN {X 0,Y 241.808,Z 624.502,A -85,B 0,C 180,E1 -21743.429,E2 -21743.429} C_VEL
LIN {X 0,Y 235.159,Z 631.313,A -85,B 0,C 180,E1 -21745.4,E2 -21745.4} C_VEL
LIN {X 0,Y 228.932,Z 636.855,A -85,B 0,C 180,E1 -21747.505,E2 -21747.505} C_VEL
LIN {X 0,Y 221.194,Z 642.613,A -85,B 0,C 180,E1 -21750.496,E2 -21750.496} C_VEL
LIN {X 0,Y 215.927,Z 645.8,A -85,B 0,C 180,E1 -21752.892,E2 -21752.892} C_VEL
LIN {X 0,Y 209.519,Z 648.712,A -85,B 0,C 180,E1 -21756.264,E2 -21756.264} C_VEL
LIN {X 0,Y 203.908,Z 650.062,A -85,B 0,C 180,E1 -21759.839,E2 -21759.839} C_VEL
LIN {X 0,Y 199.332,Z 649.935,A -85,B 0,C 180,E1 -21763.617,E2 -21763.617} C_VEL
LIN {X 0,Y 195.849,Z 648.263,A -85,B 0,C 180,E1 -21767.566,E2 -21767.566} C_VEL
LIN {X 0,Y 193.382,Z 645.065,A -85,B 0,C 180,E1 -21771.641,E2 -21771.641} C_VEL
LIN {X 0,Y 192.057,Z 641.627,A -85,B 0,C 180,E1 -21774.751,E2 -21774.751} C_VEL
LIN {X 0,Y 191.249,Z 637.197,A -85,B 0,C 180,E1 -21777.894,E2 -21777.894} C_VEL
LIN {X 0,Y 191.032,Z 630.672,A -85,B 0,C 180,E1 -21781.581,E2 -21781.581} C_VEL
LIN {X 0,Y 191.367,Z 623.751,A -85,B 0,C 180,E1 -21784.74,E2 -21784.74} C_VEL
LIN {X 0,Y 191.699,Z 615.318,A -85,B 0,C 180,E1 -21787.857,E2 -21787.857} C_VEL
LIN {X 0,Y 192.393,Z 604.666,A -85,B 0,C 180,E1 -21791.057,E2 -21791.057} C_VEL
LIN {X 0,Y 193.396,Z 592.749,A -85,B 0,C 180,E1 -21793.931,E2 -21793.931} C_VEL
LIN {X 0,Y 194.405,Z 580.699,A -85,B 0,C 180,E1 -21796.271,E2 -21796.271} C_VEL
LIN {X 0,Y 195.505,Z 567.405,A -85,B 0,C 180,E1 -21798.334,E2 -21798.334} C_VEL
LIN {X 0,Y 196.317,Z 554.404,A -85,B 0,C 180,E1 -21799.883,E2 -21799.883} C_VEL
LIN {X 0,Y 197.139,Z 539.983,A -85,B 0,C 180,E1 -21801.15,E2 -21801.15} C_VEL
LIN {X 0,Y 199.835,Z 475.808,A -85,B 0,C 180,E1 -21805.222,E2 -21805.222} C_VEL
LIN {X 0,Y 193.181,Z 451.651,A -85,B 0,C 180,E1 -21807.034,E2 -21807.034} C_VEL
LIN {X 0,Y 192.705,Z 449.47,A -85,B 0,C 180,E1 -21807.243,E2 -21807.243} C_VEL
LIN {X 0,Y 192.609,Z 449.455,A -85,B 0,C 180,E1 -21812.94,E2 -21812.94} C_VEL
LIN {X 0,Y 192.572,Z 449.621,A -85,B 0,C 180,E1 -21815.006,E2 -21815.006} C_VEL
LIN {X 0,Y 195.614,Z 456.793,A -85,B 0,C 180,E1 -21818.957,E2 -21818.957} C_VEL
LIN {X 0,Y 198.796,Z 464.813,A -85,B 0,C 180,E1 -21822.886,E2 -21822.886} C_VEL
LIN {X 0,Y 202.058,Z 474.279,A -85,B 0,C 180,E1 -21826.922,E2 -21826.922} C_VEL
LIN {X 0,Y 202.724,Z 476.343,A -85,B 0,C 180,E1 -21827.678,E2 -21827.678} C_VEL
LIN {X 0,Y 209.347,Z 488.504,A -85,B 0,C 180,E1 -21829.852,E2 -21829.852} C_VEL
LIN {X 0,Y 215.768,Z 502.539,A -85,B 0,C 180,E1 -21831.866,E2 -21831.866} C_VEL
LIN {X 0,Y 217.748,Z 507.827,A -85,B 0,C 180,E1 -21832.492,E2 -21832.492} C_VEL
LIN {X 0,Y 219.462,Z 520.262,A -85,B 0,C 180,E1 -21833.336,E2 -21833.336} C_VEL
LIN {X 0,Y 216.331,Z 585.236,A -85,B 0,C 180,E1 -21835.359,E2 -21835.359} C_VEL
LIN {X 0,Y 215.091,Z 598.804,A -85,B 0,C 180,E1 -21836.047,E2 -21836.047} C_VEL
LIN {X 0,Y 213.452,Z 610.473,A -85,B 0,C 180,E1 -21836.953,E2 -21836.953} C_VEL
LIN {X 0,Y 211.462,Z 621.636,A -85,B 0,C 180,E1 -21838.156,E2 -21838.156} C_VEL
LIN {X 0,Y 208.989,Z 632.63,A -85,B 0,C 180,E1 -21839.706,E2 -21839.706} C_VEL
LIN {X 0,Y 205.991,Z 643.839,A -85,B 0,C 180,E1 -21841.745,E2 -21841.745} C_VEL
LIN {X 0,Y 203.439,Z 652.712,A -85,B 0,C 180,E1 -21843.813,E2 -21843.813} C_VEL
LIN {X 0,Y 200.764,Z 661.151,A -85,B 0,C 180,E1 -21846.261,E2 -21846.261} C_VEL
LIN {X 0,Y 197.813,Z 669.203,A -85,B 0,C 180,E1 -21849.189,E2 -21849.189} C_VEL
LIN {X 0,Y 195.427,Z 675.674,A -85,B 0,C 180,E1 -21852.201,E2 -21852.201} C_VEL
LIN {X 0,Y 193.54,Z 680.815,A -85,B 0,C 180,E1 -21855.274,E2 -21855.274} C_VEL
LIN {X 0,Y 192.097,Z 684.792,A -85,B 0,C 180,E1 -21858.392,E2 -21858.392} C_VEL
LIN {X 0,Y 191.123,Z 687.72,A -85,B 0,C 180,E1 -21861.542,E2 -21861.542} C_VEL
LIN {X 0,Y 190.529,Z 689.754,A -85,B 0,C 180,E1 -21864.841,E2 -21864.841} C_VEL
LIN {X 0,Y 190.29,Z 690.739,A -85,B 0,C 180,E1 -21867.883,E2 -21867.883} C_VEL
LIN {X 0,Y 190.282,Z 690.968,A -85,B 0,C 180,E1 -21870,E2 -21870} C_VEL
LIN {X 0,Y 190.29,Z 690.771,A -85,B 0,C 180,E1 -21872.117,E2 -21872.117} C_VEL
LIN {X 0,Y 190.721,Z 689.211,A -85,B 0,C 180,E1 -21876.347,E2 -21876.347} C_VEL
LIN {X 0,Y 191.118,Z 687.838,A -85,B 0,C 180,E1 -21878.459,E2 -21878.459} C_VEL
LIN {X 0,Y 192.086,Z 684.954,A -85,B 0,C 180,E1 -21881.609,E2 -21881.609} C_VEL
LIN {X 0,Y 193.483,Z 681.032,A -85,B 0,C 180,E1 -21884.73,E2 -21884.73} C_VEL
LIN {X 0,Y 195.394,Z 675.945,A -85,B 0,C 180,E1 -21887.802,E2 -21887.802} C_VEL
LIN {X 0,Y 197.787,Z 669.529,A -85,B 0,C 180,E1 -21890.814,E2 -21890.814} C_VEL
LIN {X 0,Y 200.691,Z 661.553,A -85,B 0,C 180,E1 -21893.748,E2 -21893.748} C_VEL
LIN {X 0,Y 203.273,Z 653.429,A -85,B 0,C 180,E1 -21896.145,E2 -21896.145} C_VEL
LIN {X 0,Y 205.915,Z 644.47,A -85,B 0,C 180,E1 -21898.266,E2 -21898.266} C_VEL
LIN {X 0,Y 208.934,Z 633.389,A -85,B 0,C 180,E1 -21900.302,E2 -21900.302} C_VEL
LIN {X 0,Y 211.344,Z 622.574,A -85,B 0,C 180,E1 -21901.864,E2 -21901.864} C_VEL
LIN {X 0,Y 213.631,Z 610.59,A -85,B 0,C 180,E1 -21903.157,E2 -21903.157} C_VEL
LIN {X 0,Y 215.32,Z 597.252,A -85,B 0,C 180,E1 -21904.196,E2 -21904.196} C_VEL
LIN {X 0,Y 216.516,Z 583.945,A -85,B 0,C 180,E1 -21904.826,E2 -21904.826} C_VEL
LIN {X 0,Y 219.571,Z 520.01,A -85,B 0,C 180,E1 -21906.808,E2 -21906.808} C_VEL
LIN {X 0,Y 217.615,Z 506.866,A -85,B 0,C 180,E1 -21907.732,E2 -21907.732} C_VEL
LIN {X 0,Y 211.26,Z 492.345,A -85,B 0,C 180,E1 -21909.708,E2 -21909.708} C_VEL
LIN {X 0,Y 204.864,Z 479.992,A -85,B 0,C 180,E1 -21911.781,E2 -21911.781} C_VEL
LIN {X 0,Y 202.634,Z 476.041,A -85,B 0,C 180,E1 -21912.561,E2 -21912.561} C_VEL
LIN {X 0,Y 199.849,Z 467.748,A -85,B 0,C 180,E1 -21916.009,E2 -21916.009} C_VEL
LIN {X 0,Y 196.956,Z 460.052,A -85,B 0,C 180,E1 -21919.625,E2 -21919.625} C_VEL
LIN {X 0,Y 193.687,Z 452.298,A -85,B 0,C 180,E1 -21923.703,E2 -21923.703} C_VEL
LIN {X 0,Y 193.058,Z 451.347,A -85,B 0,C 180,E1 -21924.326,E2 -21924.326} C_VEL
LIN {X 0,Y 196.242,Z 466.612,A -85,B 0,C 180,E1 -21928.948,E2 -21928.948} C_VEL
LIN {X 0,Y 197.882,Z 474.737,A -85,B 0,C 180,E1 -21931.35,E2 -21931.35} C_VEL
LIN {X 0,Y 197.801,Z 476.798,A -85,B 0,C 180,E1 -21931.894,E2 -21931.894} C_VEL
LIN {X 0,Y 199.015,Z 496.492,A -85,B 0,C 180,E1 -21933.191,E2 -21933.191} C_VEL
LIN {X 0,Y 200.512,Z 512.143,A -85,B 0,C 180,E1 -21934.224,E2 -21934.224} C_VEL
LIN {X 0,Y 196.812,Z 587.844,A -85,B 0,C 180,E1 -21939.035,E2 -21939.035} C_VEL
LIN {X 0,Y 196.022,Z 601.271,A -85,B 0,C 180,E1 -21940.223,E2 -21940.223} C_VEL
LIN {X 0,Y 194.991,Z 615.13,A -85,B 0,C 180,E1 -21941.888,E2 -21941.888} C_VEL
LIN {X 0,Y 193.966,Z 628.284,A -85,B 0,C 180,E1 -21943.962,E2 -21943.962} C_VEL
LIN {X 0,Y 192.954,Z 639.931,A -85,B 0,C 180,E1 -21946.305,E2 -21946.305} C_VEL
LIN {X 0,Y 192.089,Z 650.533,A -85,B 0,C 180,E1 -21948.925,E2 -21948.925} C_VEL
LIN {X 0,Y 191.356,Z 660.831,A -85,B 0,C 180,E1 -21952.084,E2 -21952.084} C_VEL
LIN {X 0,Y 190.886,Z 669.021,A -85,B 0,C 180,E1 -21955.215,E2 -21955.215} C_VEL
LIN {X 0,Y 190.751,Z 674.756,A -85,B 0,C 180,E1 -21957.888,E2 -21957.888} C_VEL
LIN {X 0,Y 190.636,Z 680.226,A -85,B 0,C 180,E1 -21961.056,E2 -21961.056} C_VEL
LIN {X 0,Y 190.64,Z 681.414,A -85,B 0,C 180,E1 -21961.846,E2 -21961.846} C_VEL
LIN {X 0,Y 190.046,Z 683.644,A -85,B 0,C 180,E1 -21963.482,E2 -21963.482} C_VEL
LIN {X 0,Y 187.477,Z 686.526,A -85,B 0,C 180,E1 -21966.259,E2 -21966.259} C_VEL
LIN {X 0,Y 185.55,Z 688.305,A -85,B 0,C 180,E1 -21968.58,E2 -21968.58} C_VEL
LIN {X 0,Y 185.092,Z 689.467,A -85,B 0,C 180,E1 -21970.38,E2 -21970.38} C_VEL
LIN {X 0,Y 185.248,Z 689.834,A -85,B 0,C 180,E1 -21970.981,E2 -21970.981} C_VEL
LIN {X 0,Y 187.618,Z 692.084,A -85,B 0,C 180,E1 -21975.201,E2 -21975.201} C_VEL
LIN {X 0,Y 191.155,Z 692.893,A -85,B 0,C 180,E1 -21979.323,E2 -21979.323} C_VEL
LIN {X 0,Y 193.308,Z 692.771,A -85,B 0,C 180,E1 -21981.319,E2 -21981.319} C_VEL
LIN {X 0,Y 198.754,Z 691.453,A -85,B 0,C 180,E1 -21985.108,E2 -21985.108} C_VEL
LIN {X 0,Y 205.122,Z 688.663,A -85,B 0,C 180,E1 -21988.664,E2 -21988.664} C_VEL
LIN {X 0,Y 212.51,Z 684.359,A -85,B 0,C 180,E1 -21991.948,E2 -21991.948} C_VEL
LIN {X 0,Y 218.606,Z 680.01,A -85,B 0,C 180,E1 -21994.237,E2 -21994.237} C_VEL
LIN {X 0,Y 226.304,Z 673.699,A -85,B 0,C 180,E1 -21996.714,E2 -21996.714} C_VEL
LIN {X 0,Y 234.585,Z 665.759,A -85,B 0,C 180,E1 -21998.987,E2 -21998.987} C_VEL
LIN {X 0,Y 242.115,Z 657.409,A -85,B 0,C 180,E1 -22000.777,E2 -22000.777} C_VEL
LIN {X 0,Y 250.009,Z 647.4,A -85,B 0,C 180,E1 -22002.428,E2 -22002.428} C_VEL
LIN {X 0,Y 258.238,Z 635.056,A -85,B 0,C 180,E1 -22003.947,E2 -22003.947} C_VEL
LIN {X 0,Y 262.224,Z 628.23,A -85,B 0,C 180,E1 -22004.604,E2 -22004.604} C_VEL
LIN {X 0,Y 261.367,Z 629.784,A -85,B 0,C 180,E1 -22005.102,E2 -22005.102} C_VEL
LIN {X 0,Y 253.936,Z 642.106,A -85,B 0,C 180,E1 -22006.218,E2 -22006.218} C_VEL
LIN {X 0,Y 246.762,Z 652.242,A -85,B 0,C 180,E1 -22007.435,E2 -22007.435} C_VEL
LIN {X 0,Y 238.657,Z 662.345,A -85,B 0,C 180,E1 -22009.063,E2 -22009.063} C_VEL
LIN {X 0,Y 230.913,Z 670.73,A -85,B 0,C 180,E1 -22010.836,E2 -22010.836} C_VEL
LIN {X 0,Y 223.712,Z 677.725,A -85,B 0,C 180,E1 -22012.789,E2 -22012.789} C_VEL
LIN {X 0,Y 215.961,Z 684.375,A -85,B 0,C 180,E1 -22015.284,E2 -22015.284} C_VEL
LIN {X 0,Y 209.825,Z 688.984,A -85,B 0,C 180,E1 -22017.594,E2 -22017.594} C_VEL
LIN {X 0,Y 202.531,Z 693.744,A -85,B 0,C 180,E1 -22020.934,E2 -22020.934} C_VEL
LIN {X 0,Y 196.257,Z 696.937,A -85,B 0,C 180,E1 -22024.55,E2 -22024.55} C_VEL
LIN {X 0,Y 191.317,Z 698.73,A -85,B 0,C 180,E1 -22028.448,E2 -22028.448} C_VEL
LIN {X 0,Y 187.562,Z 699.157,A -85,B 0,C 180,E1 -22032.557,E2 -22032.557} C_VEL
LIN {X 0,Y 185.211,Z 698.163,A -85,B 0,C 180,E1 -22036.84,E2 -22036.84} C_VEL
LIN {X 0,Y 184.204,Z 696.654,A -85,B 0,C 180,E1 -22039.975,E2 -22039.975} C_VEL
LIN {X 0,Y 183.384,Z 699.078,A -85,B 0,C 180,E1 -22043.398,E2 -22043.398} C_VEL
LIN {X 0,Y 183.149,Z 700.699,A -85,B 0,C 180,E1 -22047.801,E2 -22047.801} C_VEL
LIN {X 0,Y 183.219,Z 700.917,A -85,B 0,C 180,E1 -22050,E2 -22050} C_VEL
LIN {X 0,Y 183.086,Z 700.36,A -85,B 0,C 180,E1 -22053.583,E2 -22053.583} C_VEL
LIN {X 0,Y 183.224,Z 699.044,A -85,B 0,C 180,E1 -22056.608,E2 -22056.608} C_VEL
LIN {X 0,Y 183.521,Z 697.603,A -85,B 0,C 180,E1 -22058.811,E2 -22058.811} C_VEL
LIN {X 0,Y 184.327,Z 694.616,A -85,B 0,C 180,E1 -22062.105,E2 -22062.105} C_VEL
LIN {X 0,Y 185.561,Z 690.567,A -85,B 0,C 180,E1 -22065.374,E2 -22065.374} C_VEL
LIN {X 0,Y 187.948,Z 684.341,A -85,B 0,C 180,E1 -22069.098,E2 -22069.098} C_VEL
LIN {X 0,Y 190.531,Z 677.326,A -85,B 0,C 180,E1 -22072.32,E2 -22072.32} C_VEL
LIN {X 0,Y 192.736,Z 671.091,A -85,B 0,C 180,E1 -22074.649,E2 -22074.649} C_VEL
LIN {X 0,Y 198.329,Z 667.591,A -85,B 0,C 180,E1 -22078.58,E2 -22078.58} C_VEL
LIN {X 0,Y 203.263,Z 664.112,A -85,B 0,C 180,E1 -22081.241,E2 -22081.241} C_VEL
LIN {X 0,Y 210.875,Z 658.217,A -85,B 0,C 180,E1 -22084.512,E2 -22084.512} C_VEL
LIN {X 0,Y 218.452,Z 651.705,A -85,B 0,C 180,E1 -22087.101,E2 -22087.101} C_VEL
LIN {X 0,Y 226.698,Z 643.769,A -85,B 0,C 180,E1 -22089.46,E2 -22089.46} C_VEL
LIN {X 0,Y 235.412,Z 634.503,A -85,B 0,C 180,E1 -22091.475,E2 -22091.475} C_VEL
LIN {X 0,Y 244.007,Z 624.193,A -85,B 0,C 180,E1 -22093.162,E2 -22093.162} C_VEL
LIN {X 0,Y 252.025,Z 613.258,A -85,B 0,C 180,E1 -22094.478,E2 -22094.478} C_VEL
LIN {X 0,Y 259.822,Z 601.091,A -85,B 0,C 180,E1 -22095.597,E2 -22095.597} C_VEL
LIN {X 0,Y 264.027,Z 593.593,A -85,B 0,C 180,E1 -22096.137,E2 -22096.137} C_VEL
LIN {X 0,Y 264.663,Z 592.372,A -85,B 0,C 180,E1 -22096.337,E2 -22096.337} C_VEL
LIN {X 0,Y 258.008,Z 603.172,A -85,B 0,C 180,E1 -22097.61,E2 -22097.61} C_VEL
LIN {X 0,Y 250.387,Z 613.627,A -85,B 0,C 180,E1 -22099.209,E2 -22099.209} C_VEL
LIN {X 0,Y 242.761,Z 622.597,A -85,B 0,C 180,E1 -22100.974,E2 -22100.974} C_VEL
LIN {X 0,Y 234.404,Z 630.929,A -85,B 0,C 180,E1 -22103.155,E2 -22103.155} C_VEL
LIN {X 0,Y 227.66,Z 636.714,A -85,B 0,C 180,E1 -22105.173,E2 -22105.173} C_VEL
LIN {X 0,Y 221.361,Z 641.377,A -85,B 0,C 180,E1 -22107.334,E2 -22107.334} C_VEL
LIN {X 0,Y 215.393,Z 645.102,A -85,B 0,C 180,E1 -22109.619,E2 -22109.619} C_VEL
LIN {X 0,Y 209.901,Z 647.901,A -85,B 0,C 180,E1 -22112.047,E2 -22112.047} C_VEL
LIN {X 0,Y 203.207,Z 650.307,A -85,B 0,C 180,E1 -22115.479,E2 -22115.479} C_VEL
LIN {X 0,Y 197.349,Z 651.238,A -85,B 0,C 180,E1 -22119.138,E2 -22119.138} C_VEL
LIN {X 0,Y 192.574,Z 650.641,A -85,B 0,C 180,E1 -22123.025,E2 -22123.025} C_VEL
LIN {X 0,Y 188.933,Z 648.585,A -85,B 0,C 180,E1 -22127.104,E2 -22127.104} C_VEL
LIN {X 0,Y 186.369,Z 644.984,A -85,B 0,C 180,E1 -22131.324,E2 -22131.324} C_VEL
LIN {X 0,Y 184.659,Z 639.768,A -85,B 0,C 180,E1 -22135.635,E2 -22135.635} C_VEL
LIN {X 0,Y 184.054,Z 634.695,A -85,B 0,C 180,E1 -22138.906,E2 -22138.906} C_VEL
LIN {X 0,Y 184.085,Z 627.275,A -85,B 0,C 180,E1 -22142.735,E2 -22142.735} C_VEL
LIN {X 0,Y 184.392,Z 620.847,A -85,B 0,C 180,E1 -22145.468,E2 -22145.468} C_VEL
LIN {X 0,Y 184.834,Z 611.527,A -85,B 0,C 180,E1 -22148.748,E2 -22148.748} C_VEL
LIN {X 0,Y 185.583,Z 601.15,A -85,B 0,C 180,E1 -22151.745,E2 -22151.745} C_VEL
LIN {X 0,Y 186.544,Z 589.452,A -85,B 0,C 180,E1 -22154.454,E2 -22154.454} C_VEL
LIN {X 0,Y 187.514,Z 578.088,A -85,B 0,C 180,E1 -22156.606,E2 -22156.606} C_VEL
LIN {X 0,Y 188.674,Z 563.802,A -85,B 0,C 180,E1 -22158.74,E2 -22158.74} C_VEL
LIN {X 0,Y 189.468,Z 549.486,A -85,B 0,C 180,E1 -22160.35,E2 -22160.35} C_VEL
LIN {X 0,Y 190.26,Z 534.829,A -85,B 0,C 180,E1 -22161.536,E2 -22161.536} C_VEL
LIN {X 0,Y 192.773,Z 476.843,A -85,B 0,C 180,E1 -22165.386,E2 -22165.386} C_VEL
LIN {X 0,Y 186.039,Z 452.117,A -85,B 0,C 180,E1 -22167.299,E2 -22167.299} C_VEL
LIN {X 0,Y 185.645,Z 450.349,A -85,B 0,C 180,E1 -22167.476,E2 -22167.476} C_VEL
LIN {X 0,Y 185.545,Z 450.443,A -85,B 0,C 180,E1 -22172.275,E2 -22172.275} C_VEL
LIN {X 0,Y 189.903,Z 460.536,A -85,B 0,C 180,E1 -22178.266,E2 -22178.266} C_VEL
LIN {X 0,Y 192.864,Z 468.158,A -85,B 0,C 180,E1 -22182.126,E2 -22182.126} C_VEL
LIN {X 0,Y 195.771,Z 476.465,A -85,B 0,C 180,E1 -22185.796,E2 -22185.796} C_VEL
LIN {X 0,Y 203.066,Z 489.428,A -85,B 0,C 180,E1 -22188.378,E2 -22188.378} C_VEL
LIN {X 0,Y 209.137,Z 502.335,A -85,B 0,C 180,E1 -22190.412,E2 -22190.412} C_VEL
LIN {X 0,Y 212.376,Z 510.666,A -85,B 0,C 180,E1 -22191.488,E2 -22191.488} C_VEL
LIN {X 0,Y 213.799,Z 521.549,A -85,B 0,C 180,E1 -22192.248,E2 -22192.248} C_VEL
LIN {X 0,Y 210.411,Z 587.352,A -85,B 0,C 180,E1 -22194.347,E2 -22194.347} C_VEL
LIN {X 0,Y 209.04,Z 600.653,A -85,B 0,C 180,E1 -22195.071,E2 -22195.071} C_VEL
LIN {X 0,Y 207.147,Z 612.868,A -85,B 0,C 180,E1 -22196.104,E2 -22196.104} C_VEL
LIN {X 0,Y 204.709,Z 625.222,A -85,B 0,C 180,E1 -22197.559,E2 -22197.559} C_VEL
LIN {X 0,Y 202.19,Z 635.573,A -85,B 0,C 180,E1 -22199.156,E2 -22199.156} C_VEL
LIN {X 0,Y 199.145,Z 646.174,A -85,B 0,C 180,E1 -22201.26,E2 -22201.26} C_VEL
LIN {X 0,Y 196.293,Z 655.159,A -85,B 0,C 180,E1 -22203.521,E2 -22203.521} C_VEL
LIN {X 0,Y 193.191,Z 664.244,A -85,B 0,C 180,E1 -22206.412,E2 -22206.412} C_VEL
LIN {X 0,Y 190.264,Z 671.714,A -85,B 0,C 180,E1 -22209.457,E2 -22209.457} C_VEL
LIN {X 0,Y 187.96,Z 677.701,A -85,B 0,C 180,E1 -22212.595,E2 -22212.595} C_VEL
LIN {X 0,Y 186.088,Z 682.433,A -85,B 0,C 180,E1 -22215.789,E2 -22215.789} C_VEL
LIN {X 0,Y 184.752,Z 686.049,A -85,B 0,C 180,E1 -22219.035,E2 -22219.035} C_VEL
LIN {X 0,Y 184.113,Z 687.909,A -85,B 0,C 180,E1 -22221.217,E2 -22221.217} C_VEL
LIN {X 0,Y 183.397,Z 690.142,A -85,B 0,C 180,E1 -22225.109,E2 -22225.109} C_VEL
LIN {X 0,Y 183.202,Z 690.928,A -85,B 0,C 180,E1 -22227.801,E2 -22227.801} C_VEL
LIN {X 0,Y 183.189,Z 691.157,A -85,B 0,C 180,E1 -22230,E2 -22230} C_VEL
LIN {X 0,Y 183.202,Z 690.96,A -85,B 0,C 180,E1 -22232.199,E2 -22232.199} C_VEL
LIN {X 0,Y 183.682,Z 689.399,A -85,B 0,C 180,E1 -22236.591,E2 -22236.591} C_VEL
LIN {X 0,Y 184.106,Z 688.026,A -85,B 0,C 180,E1 -22238.783,E2 -22238.783} C_VEL
LIN {X 0,Y 185.118,Z 685.142,A -85,B 0,C 180,E1 -22242.053,E2 -22242.053} C_VEL
LIN {X 0,Y 186.608,Z 681.219,A -85,B 0,C 180,E1 -22245.286,E2 -22245.286} C_VEL
LIN {X 0,Y 188.622,Z 676.131,A -85,B 0,C 180,E1 -22248.464,E2 -22248.464} C_VEL
LIN {X 0,Y 191.162,Z 669.714,A -85,B 0,C 180,E1 -22251.571,E2 -22251.571} C_VEL
LIN {X 0,Y 194.191,Z 661.735,A -85,B 0,C 180,E1 -22254.595,E2 -22254.595} C_VEL
LIN {X 0,Y 196.974,Z 653.424,A -85,B 0,C 180,E1 -22257.109,E2 -22257.109} C_VEL
LIN {X 0,Y 199.689,Z 644.646,A -85,B 0,C 180,E1 -22259.231,E2 -22259.231} C_VEL
LIN {X 0,Y 202.832,Z 633.561,A -85,B 0,C 180,E1 -22261.315,E2 -22261.315} C_VEL
LIN {X 0,Y 205.348,Z 622.739,A -85,B 0,C 180,E1 -22262.91,E2 -22262.91} C_VEL
LIN {X 0,Y 207.737,Z 610.742,A -85,B 0,C 180,E1 -22264.225,E2 -22264.225} C_VEL
LIN {X 0,Y 209.383,Z 598.234,A -85,B 0,C 180,E1 -22265.233,E2 -22265.233} C_VEL
LIN {X 0,Y 210.632,Z 585.44,A -85,B 0,C 180,E1 -22265.874,E2 -22265.874} C_VEL
LIN {X 0,Y 213.845,Z 520.892,A -85,B 0,C 180,E1 -22267.93,E2 -22267.93} C_VEL
LIN {X 0,Y 212.144,Z 509.368,A -85,B 0,C 180,E1 -22268.78,E2 -22268.78} C_VEL
LIN {X 0,Y 205.946,Z 495.266,A -85,B 0,C 180,E1 -22270.817,E2 -22270.817} C_VEL
LIN {X 0,Y 200.377,Z 484.449,A -85,B 0,C 180,E1 -22272.726,E2 -22272.726} C_VEL
LIN {X 0,Y 195.668,Z 476.215,A -85,B 0,C 180,E1 -22274.449,E2 -22274.449} C_VEL
LIN {X 0,Y 192.689,Z 467.649,A -85,B 0,C 180,E1 -22278.332,E2 -22278.332} C_VEL
LIN {X 0,Y 189.555,Z 459.81,A -85,B 0,C 180,E1 -22282.366,E2 -22282.366} C_VEL
LIN {X 0,Y 188.752,Z 457.881,A -85,B 0,C 180,E1 -22283.434,E2 -22283.434} C_VEL
LIN {X 0,Y 186.755,Z 455.735,A -85,B 0,C 180,E1 -22285.142,E2 -22285.142} C_VEL
LIN {X 0,Y 190.085,Z 471.67,A -85,B 0,C 180,E1 -22290.057,E2 -22290.057} C_VEL
LIN {X 0,Y 190.82,Z 476.563,A -85,B 0,C 180,E1 -22291.509,E2 -22291.509} C_VEL
LIN {X 0,Y 191.402,Z 490.202,A -85,B 0,C 180,E1 -22292.503,E2 -22292.503} C_VEL
LIN {X 0,Y 193.416,Z 513.231,A -85,B 0,C 180,E1 -22294.085,E2 -22294.085} C_VEL
LIN {X 0,Y 189.793,Z 586.806,A -85,B 0,C 180,E1 -22298.978,E2 -22298.978} C_VEL
LIN {X 0,Y 188.921,Z 601.214,A -85,B 0,C 180,E1 -22300.298,E2 -22300.298} C_VEL
LIN {X 0,Y 187.891,Z 614.958,A -85,B 0,C 180,E1 -22302.026,E2 -22302.026} C_VEL
LIN {X 0,Y 186.881,Z 628.094,A -85,B 0,C 180,E1 -22304.178,E2 -22304.178} C_VEL
LIN {X 0,Y 185.84,Z 639.798,A -85,B 0,C 180,E1 -22306.607,E2 -22306.607} C_VEL
LIN {X 0,Y 185.084,Z 649.497,A -85,B 0,C 180,E1 -22309.055,E2 -22309.055} C_VEL
LIN {X 0,Y 184.44,Z 658.634,A -85,B 0,C 180,E1 -22311.853,E2 -22311.853} C_VEL
LIN {X 0,Y 183.95,Z 667.005,A -85,B 0,C 180,E1 -22315.034,E2 -22315.034} C_VEL
LIN {X 0,Y 183.747,Z 674.145,A -85,B 0,C 180,E1 -22318.356,E2 -22318.356} C_VEL
LIN {X 0,Y 183.664,Z 680.323,A -85,B 0,C 180,E1 -22322.019,E2 -22322.019} C_VEL
LIN {X 0,Y 183.748,Z 684.295,A -85,B 0,C 180,E1 -22325.012,E2 -22325.012} C_VEL
LIN {X 0,Y 184.501,Z 688.111,A -85,B 0,C 180,E1 -22328.764,E2 -22328.764} C_VEL
LIN {X 0,Y 185.248,Z 689.834,A -85,B 0,C 180,E1 -22330.981,E2 -22330.981} C_VEL
LIN {X 0,Y 185.439,Z 690.896,A -85,B 0,C 180,E1 -22332.781,E2 -22332.781} C_VEL
LIN {X 0,Y 184.447,Z 692.141,A -85,B 0,C 180,E1 -22335.813,E2 -22335.813} C_VEL
LIN {X 0,Y 184.047,Z 692.927,A -85,B 0,C 180,E1 -22338.879,E2 -22338.879} C_VEL
LIN {X 0,Y 185.141,Z 693.129,A -85,B 0,C 180,E1 -22340.677,E2 -22340.677} C_VEL
LIN {X 0,Y 189.467,Z 692.957,A -85,B 0,C 180,E1 -22344.081,E2 -22344.081} C_VEL
LIN {X 0,Y 195.617,Z 691.354,A -85,B 0,C 180,E1 -22347.843,E2 -22347.843} C_VEL
LIN {X 0,Y 202.73,Z 688.372,A -85,B 0,C 180,E1 -22351.332,E2 -22351.332} C_VEL
LIN {X 0,Y 210.883,Z 683.822,A -85,B 0,C 180,E1 -22354.51,E2 -22354.51} C_VEL
LIN {X 0,Y 219.85,Z 677.591,A -85,B 0,C 180,E1 -22357.4,E2 -22357.4} C_VEL
LIN {X 0,Y 227.28,Z 671.541,A -85,B 0,C 180,E1 -22359.453,E2 -22359.453} C_VEL
LIN {X 0,Y 236.63,Z 662.639,A -85,B 0,C 180,E1 -22361.648,E2 -22361.648} C_VEL
LIN {X 0,Y 244.047,Z 654.436,A -85,B 0,C 180,E1 -22363.17,E2 -22363.17} C_VEL
LIN {X 0,Y 250.984,Z 645.781,A -85,B 0,C 180,E1 -22364.431,E2 -22364.431} C_VEL
LIN {X 0,Y 251.237,Z 645.46,A -85,B 0,C 180,E1 -22364.867,E2 -22364.867} C_VEL
LIN {X 0,Y 243.384,Z 655.551,A -85,B 0,C 180,E1 -22366.129,E2 -22366.129} C_VEL
LIN {X 0,Y 235.004,Z 664.92,A -85,B 0,C 180,E1 -22367.71,E2 -22367.71} C_VEL
LIN {X 0,Y 227.011,Z 672.827,A -85,B 0,C 180,E1 -22369.448,E2 -22369.448} C_VEL
LIN {X 0,Y 219.531,Z 679.328,A -85,B 0,C 180,E1 -22371.371,E2 -22371.371} C_VEL
LIN {X 0,Y 212.549,Z 684.766,A -85,B 0,C 180,E1 -22373.475,E2 -22373.475} C_VEL
LIN {X 0,Y 203.978,Z 690.472,A -85,B 0,C 180,E1 -22376.545,E2 -22376.545} C_VEL
LIN {X 0,Y 196.419,Z 694.633,A -85,B 0,C 180,E1 -22379.938,E2 -22379.938} C_VEL
LIN {X 0,Y 189.883,Z 697.364,A -85,B 0,C 180,E1 -22383.631,E2 -22383.631} C_VEL
LIN {X 0,Y 184.747,Z 698.689,A -85,B 0,C 180,E1 -22387.641,E2 -22387.641} C_VEL
LIN {X 0,Y 180.8,Z 698.683,A -85,B 0,C 180,E1 -22391.882,E2 -22391.882} C_VEL
LIN {X 0,Y 178.34,Z 697.343,A -85,B 0,C 180,E1 -22396.323,E2 -22396.323} C_VEL
LIN {X 0,Y 177.425,Z 695.986,A -85,B 0,C 180,E1 -22399.01,E2 -22399.01} C_VEL
LIN {X 0,Y 176.332,Z 698.889,A -85,B 0,C 180,E1 -22403.133,E2 -22403.133} C_VEL
LIN {X 0,Y 176.046,Z 700.51,A -85,B 0,C 180,E1 -22407.712,E2 -22407.712} C_VEL
LIN {X 0,Y 176.125,Z 700.728,A -85,B 0,C 180,E1 -22410,E2 -22410} C_VEL
LIN {X 0,Y 175.996,Z 700.277,A -85,B 0,C 180,E1 -22413.319,E2 -22413.319} C_VEL
LIN {X 0,Y 176.15,Z 698.854,A -85,B 0,C 180,E1 -22416.874,E2 -22416.874} C_VEL
LIN {X 0,Y 176.481,Z 697.412,A -85,B 0,C 180,E1 -22419.166,E2 -22419.166} C_VEL
LIN {X 0,Y 177.355,Z 694.426,A -85,B 0,C 180,E1 -22422.589,E2 -22422.589} C_VEL
LIN {X 0,Y 178.694,Z 690.377,A -85,B 0,C 180,E1 -22425.981,E2 -22425.981} C_VEL
LIN {X 0,Y 181.203,Z 684.151,A -85,B 0,C 180,E1 -22429.839,E2 -22429.839} C_VEL
LIN {X 0,Y 183.834,Z 677.425,A -85,B 0,C 180,E1 -22433.039,E2 -22433.039} C_VEL
LIN {X 0,Y 186.379,Z 670.74,A -85,B 0,C 180,E1 -22435.624,E2 -22435.624} C_VEL
LIN {X 0,Y 190.55,Z 668.57,A -85,B 0,C 180,E1 -22438.651,E2 -22438.651} C_VEL
LIN {X 0,Y 197.244,Z 664.631,A -85,B 0,C 180,E1 -22442.308,E2 -22442.308} C_VEL
LIN {X 0,Y 205.131,Z 659.315,A -85,B 0,C 180,E1 -22445.622,E2 -22445.622} C_VEL
LIN {X 0,Y 214.116,Z 652.397,A -85,B 0,C 180,E1 -22448.583,E2 -22448.583} C_VEL
LIN {X 0,Y 222.667,Z 644.977,A -85,B 0,C 180,E1 -22450.914,E2 -22450.914} C_VEL
LIN {X 0,Y 232.049,Z 635.92,A -85,B 0,C 180,E1 -22452.965,E2 -22452.965} C_VEL
LIN {X 0,Y 241.964,Z 624.916,A -85,B 0,C 180,E1 -22454.778,E2 -22454.778} C_VEL
LIN {X 0,Y 250.263,Z 614.466,A -85,B 0,C 180,E1 -22456.023,E2 -22456.023} C_VEL
LIN {X 0,Y 252.566,Z 611.267,A -85,B 0,C 180,E1 -22456.343,E2 -22456.343} C_VEL
LIN {X 0,Y 253.443,Z 609.933,A -85,B 0,C 180,E1 -22456.767,E2 -22456.767} C_VEL
LIN {X 0,Y 245.696,Z 619.213,A -85,B 0,C 180,E1 -22458.313,E2 -22458.313} C_VEL
LIN {X 0,Y 237.948,Z 627.227,A -85,B 0,C 180,E1 -22460.029,E2 -22460.029} C_VEL
LIN {X 0,Y 229.304,Z 634.808,A -85,B 0,C 180,E1 -22462.194,E2 -22462.194} C_VEL
LIN {X 0,Y 222.361,Z 640.019,A -85,B 0,C 180,E1 -22464.217,E2 -22464.217} C_VEL
LIN {X 0,Y 213.697,Z 645.439,A -85,B 0,C 180,E1 -22467.136,E2 -22467.136} C_VEL
LIN {X 0,Y 207.649,Z 648.417,A -85,B 0,C 180,E1 -22469.49,E2 -22469.49} C_VEL
LIN {X 0,Y 200.304,Z 651.041,A -85,B 0,C 180,E1 -22472.863,E2 -22472.863} C_VEL
LIN {X 0,Y 193.762,Z 652.215,A -85,B 0,C 180,E1 -22476.485,E2 -22476.485} C_VEL
LIN {X 0,Y 188.212,Z 651.955,A -85,B 0,C 180,E1 -22480.363,E2 -22480.363} C_VEL
LIN {X 0,Y 183.769,Z 650.181,A -85,B 0,C 180,E1 -22484.472,E2 -22484.472} C_VEL
LIN {X 0,Y 180.576,Z 646.951,A -85,B 0,C 180,E1 -22488.779,E2 -22488.779} C_VEL
LIN {X 0,Y 178.832,Z 643.506,A -85,B 0,C 180,E1 -22492.094,E2 -22492.094} C_VEL
LIN {X 0,Y 177.603,Z 639.105,A -85,B 0,C 180,E1 -22495.461,E2 -22495.461} C_VEL
LIN {X 0,Y 176.976,Z 632.665,A -85,B 0,C 180,E1 -22499.431,E2 -22499.431} C_VEL
LIN {X 0,Y 177.167,Z 624.637,A -85,B 0,C 180,E1 -22503.411,E2 -22503.411} C_VEL
LIN {X 0,Y 177.421,Z 617.565,A -85,B 0,C 180,E1 -22506.254,E2 -22506.254} C_VEL
LIN {X 0,Y 178.016,Z 607.359,A -85,B 0,C 180,E1 -22509.659,E2 -22509.659} C_VEL
LIN {X 0,Y 178.902,Z 595.873,A -85,B 0,C 180,E1 -22512.766,E2 -22512.766} C_VEL
LIN {X 0,Y 179.85,Z 584.413,A -85,B 0,C 180,E1 -22515.294,E2 -22515.294} C_VEL
LIN {X 0,Y 180.711,Z 573.472,A -85,B 0,C 180,E1 -22517.25,E2 -22517.25} C_VEL
LIN {X 0,Y 181.803,Z 559.783,A -85,B 0,C 180,E1 -22519.183,E2 -22519.183} C_VEL
LIN {X 0,Y 182.634,Z 545.385,A -85,B 0,C 180,E1 -22520.705,E2 -22520.705} C_VEL
LIN {X 0,Y 183.42,Z 528.082,A -85,B 0,C 180,E1 -22522.011,E2 -22522.011} C_VEL
LIN {X 0,Y 185.684,Z 477.834,A -85,B 0,C 180,E1 -22525.524,E2 -22525.524} C_VEL
LIN {X 0,Y 178.914,Z 452.744,A -85,B 0,C 180,E1 -22527.523,E2 -22527.523} C_VEL
LIN {X 0,Y 178.621,Z 451.223,A -85,B 0,C 180,E1 -22527.691,E2 -22527.691} C_VEL
LIN {X 0,Y 178.574,Z 451.367,A -85,B 0,C 180,E1 -22529.168,E2 -22529.168} C_VEL
LIN {X 0,Y 179.242,Z 453.645,A -85,B 0,C 180,E1 -22530.646,E2 -22530.646} C_VEL
LIN {X 0,Y 180.197,Z 455.006,A -85,B 0,C 180,E1 -22531.771,E2 -22531.771} C_VEL
LIN {X 0,Y 183.831,Z 463.445,A -85,B 0,C 180,E1 -22537.015,E2 -22537.015} C_VEL
LIN {X 0,Y 186.918,Z 471.334,A -85,B 0,C 180,E1 -22541.237,E2 -22541.237} C_VEL
LIN {X 0,Y 188.853,Z 476.737,A -85,B 0,C 180,E1 -22543.726,E2 -22543.726} C_VEL
LIN {X 0,Y 194.598,Z 486.488,A -85,B 0,C 180,E1 -22545.966,E2 -22545.966} C_VEL
LIN {X 0,Y 199.857,Z 496.478,A -85,B 0,C 180,E1 -22547.889,E2 -22547.889} C_VEL
LIN {X 0,Y 205.856,Z 509.982,A -85,B 0,C 180,E1 -22549.993,E2 -22549.993} C_VEL
LIN {X 0,Y 207.013,Z 513.321,A -85,B 0,C 180,E1 -22550.41,E2 -22550.41} C_VEL
LIN {X 0,Y 208.182,Z 522.982,A -85,B 0,C 180,E1 -22551.099,E2 -22551.099} C_VEL
LIN {X 0,Y 204.718,Z 586.978,A -85,B 0,C 180,E1 -22553.167,E2 -22553.167} C_VEL
LIN {X 0,Y 203.377,Z 600.08,A -85,B 0,C 180,E1 -22553.881,E2 -22553.881} C_VEL
LIN {X 0,Y 201.531,Z 611.959,A -85,B 0,C 180,E1 -22554.872,E2 -22554.872} C_VEL
LIN {X 0,Y 199.176,Z 623.693,A -85,B 0,C 180,E1 -22556.238,E2 -22556.238} C_VEL
LIN {X 0,Y 196.142,Z 635.754,A -85,B 0,C 180,E1 -22558.095,E2 -22558.095} C_VEL
LIN {X 0,Y 192.958,Z 646.359,A -85,B 0,C 180,E1 -22560.247,E2 -22560.247} C_VEL
LIN {X 0,Y 189.792,Z 655.855,A -85,B 0,C 180,E1 -22562.714,E2 -22562.714} C_VEL
LIN {X 0,Y 186.705,Z 664.431,A -85,B 0,C 180,E1 -22565.539,E2 -22565.539} C_VEL
LIN {X 0,Y 183.641,Z 671.902,A -85,B 0,C 180,E1 -22568.68,E2 -22568.68} C_VEL
LIN {X 0,Y 181.173,Z 677.89,A -85,B 0,C 180,E1 -22571.921,E2 -22571.921} C_VEL
LIN {X 0,Y 179.198,Z 682.623,A -85,B 0,C 180,E1 -22575.231,E2 -22575.231} C_VEL
LIN {X 0,Y 177.786,Z 686.238,A -85,B 0,C 180,E1 -22578.6,E2 -22578.6} C_VEL
LIN {X 0,Y 177.093,Z 688.099,A -85,B 0,C 180,E1 -22580.866,E2 -22580.866} C_VEL
LIN {X 0,Y 176.635,Z 689.513,A -85,B 0,C 180,E1 -22583.145,E2 -22583.145} C_VEL
LIN {X 0,Y 176.118,Z 691.117,A -85,B 0,C 180,E1 -22587.713,E2 -22587.713} C_VEL
LIN {X 0,Y 176.099,Z 691.346,A -85,B 0,C 180,E1 -22590,E2 -22590} C_VEL
LIN {X 0,Y 176.118,Z 691.149,A -85,B 0,C 180,E1 -22592.287,E2 -22592.287} C_VEL
LIN {X 0,Y 176.635,Z 689.587,A -85,B 0,C 180,E1 -22596.855,E2 -22596.855} C_VEL
LIN {X 0,Y 177.086,Z 688.214,A -85,B 0,C 180,E1 -22599.134,E2 -22599.134} C_VEL
LIN {X 0,Y 178.174,Z 685.33,A -85,B 0,C 180,E1 -22602.53,E2 -22602.53} C_VEL
LIN {X 0,Y 179.76,Z 681.406,A -85,B 0,C 180,E1 -22605.883,E2 -22605.883} C_VEL
LIN {X 0,Y 181.889,Z 676.317,A -85,B 0,C 180,E1 -22609.174,E2 -22609.174} C_VEL
LIN {X 0,Y 184.575,Z 669.898,A -85,B 0,C 180,E1 -22612.381,E2 -22612.381} C_VEL
LIN {X 0,Y 187.744,Z 661.918,A -85,B 0,C 180,E1 -22615.499,E2 -22615.499} C_VEL
LIN {X 0,Y 190.63,Z 653.732,A -85,B 0,C 180,E1 -22618.046,E2 -22618.046} C_VEL
LIN {X 0,Y 193.538,Z 644.822,A -85,B 0,C 180,E1 -22620.255,E2 -22620.255} C_VEL
LIN {X 0,Y 196.816,Z 633.731,A -85,B 0,C 180,E1 -22622.387,E2 -22622.387} C_VEL
LIN {X 0,Y 199.438,Z 622.903,A -85,B 0,C 180,E1 -22624.016,E2 -22624.016} C_VEL
LIN {X 0,Y 201.922,Z 610.894,A -85,B 0,C 180,E1 -22625.355,E2 -22625.355} C_VEL
LIN {X 0,Y 203.634,Z 598.449,A -85,B 0,C 180,E1 -22626.376,E2 -22626.376} C_VEL
LIN {X 0,Y 204.912,Z 585.926,A -85,B 0,C 180,E1 -22627.016,E2 -22627.016} C_VEL
LIN {X 0,Y 208.255,Z 522.111,A -85,B 0,C 180,E1 -22629.087,E2 -22629.087} C_VEL
LIN {X 0,Y 206.93,Z 512.435,A -85,B 0,C 180,E1 -22629.815,E2 -22629.815} C_VEL
LIN {X 0,Y 201.222,Z 499.315,A -85,B 0,C 180,E1 -22631.801,E2 -22631.801} C_VEL
LIN {X 0,Y 196.141,Z 489.18,A -85,B 0,C 180,E1 -22633.646,E2 -22633.646} C_VEL
LIN {X 0,Y 190.223,Z 479.022,A -85,B 0,C 180,E1 -22635.913,E2 -22635.913} C_VEL
LIN {X 0,Y 188.679,Z 476.261,A -85,B 0,C 180,E1 -22636.624,E2 -22636.624} C_VEL
LIN {X 0,Y 185.693,Z 468.059,A -85,B 0,C 180,E1 -22640.658,E2 -22640.658} C_VEL
LIN {X 0,Y 183.627,Z 462.931,A -85,B 0,C 180,E1 -22643.489,E2 -22643.489} C_VEL
LIN {X 0,Y 182.264,Z 461.474,A -85,B 0,C 180,E1 -22644.662,E2 -22644.662} C_VEL
LIN {X 0,Y 180.589,Z 460.565,A -85,B 0,C 180,E1 -22645.801,E2 -22645.801} C_VEL
LIN {X 0,Y 180.48,Z 460.298,A -85,B 0,C 180,E1 -22646.08,E2 -22646.08} C_VEL
LIN {X 0,Y 183.728,Z 476.052,A -85,B 0,C 180,E1 -22651.005,E2 -22651.005} C_VEL
LIN {X 0,Y 183.758,Z 477.03,A -85,B 0,C 180,E1 -22651.291,E2 -22651.291} C_VEL
LIN {X 0,Y 184.802,Z 495.972,A -85,B 0,C 180,E1 -22652.636,E2 -22652.636} C_VEL
LIN {X 0,Y 186.362,Z 512.9,A -85,B 0,C 180,E1 -22653.848,E2 -22653.848} C_VEL
LIN {X 0,Y 182.645,Z 587.081,A -85,B 0,C 180,E1 -22659.076,E2 -22659.076} C_VEL
LIN {X 0,Y 181.855,Z 600.86,A -85,B 0,C 180,E1 -22660.382,E2 -22660.382} C_VEL
LIN {X 0,Y 180.815,Z 614.705,A -85,B 0,C 180,E1 -22662.176,E2 -22662.176} C_VEL
LIN {X 0,Y 179.794,Z 627.898,A -85,B 0,C 180,E1 -22664.411,E2 -22664.411} C_VEL
LIN {X 0,Y 178.868,Z 638.503,A -85,B 0,C 180,E1 -22666.653,E2 -22666.653} C_VEL
LIN {X 0,Y 178.116,Z 648.293,A -85,B 0,C 180,E1 -22669.197,E2 -22669.197} C_VEL
LIN {X 0,Y 177.452,Z 657.779,A -85,B 0,C 180,E1 -22672.175,E2 -22672.175} C_VEL
LIN {X 0,Y 176.971,Z 666.242,A -85,B 0,C 180,E1 -22675.444,E2 -22675.444} C_VEL
LIN {X 0,Y 176.794,Z 673.473,A -85,B 0,C 180,E1 -22678.861,E2 -22678.861} C_VEL
LIN {X 0,Y 176.707,Z 679.195,A -85,B 0,C 180,E1 -22682.279,E2 -22682.279} C_VEL
LIN {X 0,Y 176.778,Z 683.179,A -85,B 0,C 180,E1 -22685.237,E2 -22685.237} C_VEL
LIN {X 0,Y 177.544,Z 687.327,A -85,B 0,C 180,E1 -22689.11,E2 -22689.11} C_VEL
LIN {X 0,Y 179.358,Z 690.725,A -85,B 0,C 180,E1 -22693.598,E2 -22693.598} C_VEL
LIN {X 0,Y 182.516,Z 692.65,A -85,B 0,C 180,E1 -22697.942,E2 -22697.942} C_VEL
LIN {X 0,Y 185.141,Z 693.129,A -85,B 0,C 180,E1 -22700.677,E2 -22700.677} C_VEL
LIN {X 0,Y 186.492,Z 693.232,A -85,B 0,C 180,E1 -22702.453,E2 -22702.453} C_VEL
LIN {X 0,Y 188.897,Z 692.607,A -85,B 0,C 180,E1 -22707.841,E2 -22707.841} C_VEL
LIN {X 0,Y 191.267,Z 691.873,A -85,B 0,C 180,E1 -22709.766,E2 -22709.766} C_VEL
LIN {X 0,Y 191.745,Z 691.673,A -85,B 0,C 180,E1 -22710.019,E2 -22710.019} C_VEL
LIN {X 0,Y 196.838,Z 689.896,A -85,B 0,C 180,E1 -22712.382,E2 -22712.382} C_VEL
LIN {X 0,Y 203.083,Z 687.064,A -85,B 0,C 180,E1 -22714.821,E2 -22714.821} C_VEL
LIN {X 0,Y 212.179,Z 681.914,A -85,B 0,C 180,E1 -22717.79,E2 -22717.79} C_VEL
LIN {X 0,Y 221.935,Z 675.101,A -85,B 0,C 180,E1 -22720.478,E2 -22720.478} C_VEL
LIN {X 0,Y 229.807,Z 668.667,A -85,B 0,C 180,E1 -22722.284,E2 -22722.284} C_VEL
LIN {X 0,Y 239.396,Z 659.504,A -85,B 0,C 180,E1 -22724.206,E2 -22724.206} C_VEL
LIN {X 0,Y 240.809,Z 658.042,A -85,B 0,C 180,E1 -22724.462,E2 -22724.462} C_VEL
LIN {X 0,Y 239.837,Z 659.104,A -85,B 0,C 180,E1 -22724.838,E2 -22724.838} C_VEL
LIN {X 0,Y 230.091,Z 668.855,A -85,B 0,C 180,E1 -22726.587,E2 -22726.587} C_VEL
LIN {X 0,Y 221.904,Z 675.937,A -85,B 0,C 180,E1 -22728.31,E2 -22728.31} C_VEL
LIN {X 0,Y 214.245,Z 681.862,A -85,B 0,C 180,E1 -22730.233,E2 -22730.233} C_VEL
LIN {X 0,Y 204.741,Z 688.132,A -85,B 0,C 180,E1 -22733.079,E2 -22733.079} C_VEL
LIN {X 0,Y 198.182,Z 691.8,A -85,B 0,C 180,E1 -22735.431,E2 -22735.431} C_VEL
LIN {X 0,Y 190.353,Z 695.41,A -85,B 0,C 180,E1 -22738.876,E2 -22738.876} C_VEL
LIN {X 0,Y 183.56,Z 697.654,A -85,B 0,C 180,E1 -22742.648,E2 -22742.648} C_VEL
LIN {X 0,Y 178.201,Z 698.531,A -85,B 0,C 180,E1 -22746.772,E2 -22746.772} C_VEL
LIN {X 0,Y 174.077,Z 698.08,A -85,B 0,C 180,E1 -22751.156,E2 -22751.156} C_VEL
LIN {X 0,Y 171.511,Z 696.343,A -85,B 0,C 180,E1 -22755.767,E2 -22755.767} C_VEL
LIN {X 0,Y 170.689,Z 695.269,A -85,B 0,C 180,E1 -22757.969,E2 -22757.969} C_VEL
LIN {X 0,Y 169.803,Z 697.281,A -85,B 0,C 180,E1 -22760.47,E2 -22760.47} C_VEL
LIN {X 0,Y 169.278,Z 698.701,A -85,B 0,C 180,E1 -22762.845,E2 -22762.845} C_VEL
LIN {X 0,Y 168.947,Z 700.321,A -85,B 0,C 180,E1 -22767.616,E2 -22767.616} C_VEL
LIN {X 0,Y 169.032,Z 700.539,A -85,B 0,C 180,E1 -22770,E2 -22770} C_VEL
LIN {X 0,Y 168.91,Z 700.173,A -85,B 0,C 180,E1 -22773.043,E2 -22773.043} C_VEL
LIN {X 0,Y 169.1,Z 698.665,A -85,B 0,C 180,E1 -22777.163,E2 -22777.163} C_VEL
LIN {X 0,Y 169.46,Z 697.223,A -85,B 0,C 180,E1 -22779.549,E2 -22779.549} C_VEL
LIN {X 0,Y 170.405,Z 694.236,A -85,B 0,C 180,E1 -22783.111,E2 -22783.111} C_VEL
LIN {X 0,Y 171.855,Z 690.187,A -85,B 0,C 180,E1 -22786.635,E2 -22786.635} C_VEL
LIN {X 0,Y 174.494,Z 683.961,A -85,B 0,C 180,E1 -22790.635,E2 -22790.635} C_VEL
LIN {X 0,Y 177.525,Z 676.626,A -85,B 0,C 180,E1 -22794.213,E2 -22794.213} C_VEL
LIN {X 0,Y 180.074,Z 670.251,A -85,B 0,C 180,E1 -22796.669,E2 -22796.669} C_VEL
LIN {X 0,Y 184.359,Z 668.466,A -85,B 0,C 180,E1 -22799.708,E2 -22799.708} C_VEL
LIN {X 0,Y 191.299,Z 665.024,A -85,B 0,C 180,E1 -22803.441,E2 -22803.441} C_VEL
LIN {X 0,Y 199.443,Z 660.258,A -85,B 0,C 180,E1 -22806.802,E2 -22806.802} C_VEL
LIN {X 0,Y 208.702,Z 654.002,A -85,B 0,C 180,E1 -22809.779,E2 -22809.779} C_VEL
LIN {X 0,Y 217.487,Z 647.24,A -85,B 0,C 180,E1 -22812.108,E2 -22812.108} C_VEL
LIN {X 0,Y 227.006,Z 639.037,A -85,B 0,C 180,E1 -22814.154,E2 -22814.154} C_VEL
LIN {X 0,Y 237.174,Z 629.021,A -85,B 0,C 180,E1 -22815.938,E2 -22815.938} C_VEL
LIN {X 0,Y 241.66,Z 624.128,A -85,B 0,C 180,E1 -22816.64,E2 -22816.64} C_VEL
LIN {X 0,Y 242.626,Z 622.938,A -85,B 0,C 180,E1 -22817.052,E2 -22817.052} C_VEL
LIN {X 0,Y 234.47,Z 630.533,A -85,B 0,C 180,E1 -22818.744,E2 -22818.744} C_VEL
LIN {X 0,Y 226.755,Z 636.72,A -85,B 0,C 180,E1 -22820.552,E2 -22820.552} C_VEL
LIN {X 0,Y 219.437,Z 641.75,A -85,B 0,C 180,E1 -22822.517,E2 -22822.517} C_VEL
LIN {X 0,Y 212.506,Z 645.781,A -85,B 0,C 180,E1 -22824.637,E2 -22824.637} C_VEL
LIN {X 0,Y 205.939,Z 648.927,A -85,B 0,C 180,E1 -22826.905,E2 -22826.905} C_VEL
LIN {X 0,Y 197.905,Z 651.786,A -85,B 0,C 180,E1 -22830.187,E2 -22830.187} C_VEL
LIN {X 0,Y 190.657,Z 653.198,A -85,B 0,C 180,E1 -22833.746,E2 -22833.746} C_VEL
LIN {X 0,Y 184.298,Z 653.171,A -85,B 0,C 180,E1 -22837.583,E2 -22837.583} C_VEL
LIN {X 0,Y 179.082,Z 651.717,A -85,B 0,C 180,E1 -22841.702,E2 -22841.702} C_VEL
LIN {X 0,Y 175.15,Z 648.794,A -85,B 0,C 180,E1 -22846.069,E2 -22846.069} C_VEL
LIN {X 0,Y 172.37,Z 644.369,A -85,B 0,C 180,E1 -22850.614,E2 -22850.614} C_VEL
LIN {X 0,Y 170.926,Z 639.98,A -85,B 0,C 180,E1 -22854.1,E2 -22854.1} C_VEL
LIN {X 0,Y 170.039,Z 633.566,A -85,B 0,C 180,E1 -22858.224,E2 -22858.224} C_VEL
LIN {X 0,Y 170.055,Z 625.525,A -85,B 0,C 180,E1 -22862.369,E2 -22862.369} C_VEL
LIN {X 0,Y 170.386,Z 618.623,A -85,B 0,C 180,E1 -22865.325,E2 -22865.325} C_VEL
LIN {X 0,Y 170.835,Z 608.738,A -85,B 0,C 180,E1 -22868.819,E2 -22868.819} C_VEL
LIN {X 0,Y 171.736,Z 597.22,A -85,B 0,C 180,E1 -22872.107,E2 -22872.107} C_VEL
LIN {X 0,Y 172.743,Z 584.469,A -85,B 0,C 180,E1 -22875.033,E2 -22875.033} C_VEL
LIN {X 0,Y 173.758,Z 571.704,A -85,B 0,C 180,E1 -22877.356,E2 -22877.356} C_VEL
LIN {X 0,Y 174.762,Z 558.739,A -85,B 0,C 180,E1 -22879.224,E2 -22879.224} C_VEL
LIN {X 0,Y 175.669,Z 543.29,A -85,B 0,C 180,E1 -22880.874,E2 -22880.874} C_VEL
LIN {X 0,Y 178.541,Z 478.565,A -85,B 0,C 180,E1 -22885.658,E2 -22885.658} C_VEL
LIN {X 0,Y 172.339,Z 455.664,A -85,B 0,C 180,E1 -22887.568,E2 -22887.568} C_VEL
LIN {X 0,Y 173.222,Z 456.034,A -85,B 0,C 180,E1 -22888.471,E2 -22888.471} C_VEL
LIN {X 0,Y 175.604,Z 461.169,A -85,B 0,C 180,E1 -22892.252,E2 -22892.252} C_VEL
LIN {X 0,Y 179.099,Z 469.383,A -85,B 0,C 180,E1 -22897.445,E2 -22897.445} C_VEL
LIN {X 0,Y 181.932,Z 476.858,A -85,B 0,C 180,E1 -22901.396,E2 -22901.396} C_VEL
LIN {X 0,Y 188.763,Z 488.208,A -85,B 0,C 180,E1 -22904.315,E2 -22904.315} C_VEL
LIN {X 0,Y 194.231,Z 498.367,A -85,B 0,C 180,E1 -22906.46,E2 -22906.46} C_VEL
LIN {X 0,Y 199.655,Z 510.488,A -85,B 0,C 180,E1 -22908.501,E2 -22908.501} C_VEL
LIN {X 0,Y 201.752,Z 515.917,A -85,B 0,C 180,E1 -22909.279,E2 -22909.279} C_VEL
LIN {X 0,Y 202.672,Z 523.576,A -85,B 0,C 180,E1 -22909.854,E2 -22909.854} C_VEL
LIN {X 0,Y 199.038,Z 587.865,A -85,B 0,C 180,E1 -22911.978,E2 -22911.978} C_VEL
LIN {X 0,Y 197.57,Z 601.026,A -85,B 0,C 180,E1 -22912.72,E2 -22912.72} C_VEL
LIN {X 0,Y 195.555,Z 613.21,A -85,B 0,C 180,E1 -22913.79,E2 -22913.79} C_VEL
LIN {X 0,Y 192.918,Z 625.575,A -85,B 0,C 180,E1 -22915.304,E2 -22915.304} C_VEL
LIN {X 0,Y 190.163,Z 635.935,A -85,B 0,C 180,E1 -22916.967,E2 -22916.967} C_VEL
LIN {X 0,Y 186.818,Z 646.543,A -85,B 0,C 180,E1 -22919.165,E2 -22919.165} C_VEL
LIN {X 0,Y 183.308,Z 656.599,A -85,B 0,C 180,E1 -22921.863,E2 -22921.863} C_VEL
LIN {X 0,Y 180.267,Z 664.619,A -85,B 0,C 180,E1 -22924.605,E2 -22924.605} C_VEL
LIN {X 0,Y 177.058,Z 672.09,A -85,B 0,C 180,E1 -22927.847,E2 -22927.847} C_VEL
LIN {X 0,Y 174.415,Z 678.08,A -85,B 0,C 180,E1 -22931.194,E2 -22931.194} C_VEL
LIN {X 0,Y 172.333,Z 682.813,A -85,B 0,C 180,E1 -22934.628,E2 -22934.628} C_VEL
LIN {X 0,Y 170.815,Z 686.428,A -85,B 0,C 180,E1 -22938.128,E2 -22938.128} C_VEL
LIN {X 0,Y 170.098,Z 688.288,A -85,B 0,C 180,E1 -22940.487,E2 -22940.487} C_VEL
LIN {X 0,Y 169.585,Z 689.703,A -85,B 0,C 180,E1 -22942.858,E2 -22942.858} C_VEL
LIN {X 0,Y 169.022,Z 691.306,A -85,B 0,C 180,E1 -22947.617,E2 -22947.617} C_VEL
LIN {X 0,Y 169.011,Z 691.535,A -85,B 0,C 180,E1 -22950,E2 -22950} C_VEL
LIN {X 0,Y 169.115,Z 690.954,A -85,B 0,C 180,E1 -22954.141,E2 -22954.141} C_VEL
LIN {X 0,Y 169.584,Z 689.776,A -85,B 0,C 180,E1 -22957.142,E2 -22957.142} C_VEL
LIN {X 0,Y 170.091,Z 688.402,A -85,B 0,C 180,E1 -22959.513,E2 -22959.513} C_VEL
LIN {X 0,Y 171.254,Z 685.517,A -85,B 0,C 180,E1 -22963.045,E2 -22963.045} C_VEL
LIN {X 0,Y 172.939,Z 681.593,A -85,B 0,C 180,E1 -22966.527,E2 -22966.527} C_VEL
LIN {X 0,Y 175.191,Z 676.502,A -85,B 0,C 180,E1 -22969.937,E2 -22969.937} C_VEL
LIN {X 0,Y 178.032,Z 670.082,A -85,B 0,C 180,E1 -22973.251,E2 -22973.251} C_VEL
LIN {X 0,Y 181.351,Z 662.101,A -85,B 0,C 180,E1 -22976.466,E2 -22976.466} C_VEL
LIN {X 0,Y 184.653,Z 653.117,A -85,B 0,C 180,E1 -22979.311,E2 -22979.311} C_VEL
LIN {X 0,Y 187.834,Z 643.859,A -85,B 0,C 180,E1 -22981.589,E2 -22981.589} C_VEL
LIN {X 0,Y 191.267,Z 632.52,A -85,B 0,C 180,E1 -22983.763,E2 -22983.763} C_VEL
LIN {X 0,Y 194.02,Z 621.315,A -85,B 0,C 180,E1 -22985.421,E2 -22985.421} C_VEL
LIN {X 0,Y 196.599,Z 608.575,A -85,B 0,C 180,E1 -22986.783,E2 -22986.783} C_VEL
LIN {X 0,Y 198.175,Z 597.149,A -85,B 0,C 180,E1 -22987.683,E2 -22987.683} C_VEL
LIN {X 0,Y 199.432,Z 584.214,A -85,B 0,C 180,E1 -22988.314,E2 -22988.314} C_VEL
LIN {X 0,Y 202.763,Z 523.237,A -85,B 0,C 180,E1 -22990.31,E2 -22990.31} C_VEL
LIN {X 0,Y 201.74,Z 515.464,A -85,B 0,C 180,E1 -22990.917,E2 -22990.917} C_VEL
LIN {X 0,Y 196.531,Z 503.192,A -85,B 0,C 180,E1 -22992.847,E2 -22992.847} C_VEL
LIN {X 0,Y 191.786,Z 493.618,A -85,B 0,C 180,E1 -22994.672,E2 -22994.672} C_VEL
LIN {X 0,Y 186.196,Z 483.799,A -85,B 0,C 180,E1 -22996.943,E2 -22996.943} C_VEL
LIN {X 0,Y 181.784,Z 476.565,A -85,B 0,C 180,E1 -22998.91,E2 -22998.91} C_VEL
LIN {X 0,Y 178.83,Z 468.635,A -85,B 0,C 180,E1 -23003.234,E2 -23003.234} C_VEL
LIN {X 0,Y 178.44,Z 467.747,A -85,B 0,C 180,E1 -23003.787,E2 -23003.787} C_VEL
LIN {X 0,Y 174.194,Z 464.883,A -85,B 0,C 180,E1 -23007.012,E2 -23007.012} C_VEL
LIN {X 0,Y 176.729,Z 477.439,A -85,B 0,C 180,E1 -23011.031,E2 -23011.031} C_VEL
LIN {X 0,Y 177.788,Z 496.836,A -85,B 0,C 180,E1 -23012.482,E2 -23012.482} C_VEL
LIN {X 0,Y 179.248,Z 513.773,A -85,B 0,C 180,E1 -23013.748,E2 -23013.748} C_VEL
LIN {X 0,Y 175.524,Z 587.374,A -85,B 0,C 180,E1 -23019.185,E2 -23019.185} C_VEL
LIN {X 0,Y 174.787,Z 600.504,A -85,B 0,C 180,E1 -23020.474,E2 -23020.474} C_VEL
LIN {X 0,Y 173.763,Z 614.323,A -85,B 0,C 180,E1 -23022.341,E2 -23022.341} C_VEL
LIN {X 0,Y 172.736,Z 627.448,A -85,B 0,C 180,E1 -23024.665,E2 -23024.665} C_VEL
LIN {X 0,Y 171.724,Z 639.216,A -85,B 0,C 180,E1 -23027.292,E2 -23027.292} C_VEL
LIN {X 0,Y 170.984,Z 648.906,A -85,B 0,C 180,E1 -23029.939,E2 -23029.939} C_VEL
LIN {X 0,Y 170.401,Z 657.906,A -85,B 0,C 180,E1 -23032.892,E2 -23032.892} C_VEL
LIN {X 0,Y 170.027,Z 665.365,A -85,B 0,C 180,E1 -23035.852,E2 -23035.852} C_VEL
LIN {X 0,Y 169.854,Z 672.644,A -85,B 0,C 180,E1 -23039.407,E2 -23039.407} C_VEL
LIN {X 0,Y 169.766,Z 677.653,A -85,B 0,C 180,E1 -23042.373,E2 -23042.373} C_VEL
LIN {X 0,Y 169.837,Z 682.085,A -85,B 0,C 180,E1 -23045.574,E2 -23045.574} C_VEL
LIN {X 0,Y 170.599,Z 686.394,A -85,B 0,C 180,E1 -23049.485,E2 -23049.485} C_VEL
LIN {X 0,Y 172.486,Z 690.159,A -85,B 0,C 180,E1 -23054.151,E2 -23054.151} C_VEL
LIN {X 0,Y 175.77,Z 692.516,A -85,B 0,C 180,E1 -23058.655,E2 -23058.655} C_VEL
LIN {X 0,Y 180.184,Z 693.51,A -85,B 0,C 180,E1 -23062.957,E2 -23062.957} C_VEL
LIN {X 0,Y 186.1,Z 693.077,A -85,B 0,C 180,E1 -23066.948,E2 -23066.948} C_VEL
LIN {X 0,Y 191.745,Z 691.673,A -85,B 0,C 180,E1 -23070.019,E2 -23070.019} C_VEL
LIN {X 0,Y 194.283,Z 690.828,A -85,B 0,C 180,E1 -23071.584,E2 -23071.584} C_VEL
LIN {X 0,Y 198.659,Z 688.68,A -85,B 0,C 180,E1 -23075.368,E2 -23075.368} C_VEL
LIN {X 0,Y 201.963,Z 686.894,A -85,B 0,C 180,E1 -23077.34,E2 -23077.34} C_VEL
LIN {X 0,Y 204.221,Z 685.727,A -85,B 0,C 180,E1 -23078.177,E2 -23078.177} C_VEL
LIN {X 0,Y 214.356,Z 679.936,A -85,B 0,C 180,E1 -23080.975,E2 -23080.975} C_VEL
LIN {X 0,Y 222.245,Z 674.491,A -85,B 0,C 180,E1 -23082.835,E2 -23082.835} C_VEL
LIN {X 0,Y 228.896,Z 669.365,A -85,B 0,C 180,E1 -23084.189,E2 -23084.189} C_VEL
LIN {X 0,Y 229.453,Z 668.937,A -85,B 0,C 180,E1 -23084.652,E2 -23084.652} C_VEL
LIN {X 0,Y 219.608,Z 676.869,A -85,B 0,C 180,E1 -23086.524,E2 -23086.524} C_VEL
LIN {X 0,Y 211.557,Z 682.499,A -85,B 0,C 180,E1 -23088.363,E2 -23088.363} C_VEL
LIN {X 0,Y 204,Z 687.18,A -85,B 0,C 180,E1 -23090.406,E2 -23090.406} C_VEL
LIN {X 0,Y 194.669,Z 691.998,A -85,B 0,C 180,E1 -23093.438,E2 -23093.438} C_VEL
LIN {X 0,Y 188.276,Z 694.679,A -85,B 0,C 180,E1 -23095.949,E2 -23095.949} C_VEL
LIN {X 0,Y 180.656,Z 697.069,A -85,B 0,C 180,E1 -23099.62,E2 -23099.62} C_VEL
LIN {X 0,Y 174.305,Z 698.154,A -85,B 0,C 180,E1 -23103.671,E2 -23103.671} C_VEL
LIN {X 0,Y 169.446,Z 697.961,A -85,B 0,C 180,E1 -23108.081,E2 -23108.081} C_VEL
LIN {X 0,Y 167.397,Z 697.352,A -85,B 0,C 180,E1 -23110.374,E2 -23110.374} C_VEL
LIN {X 0,Y 164.712,Z 695.221,A -85,B 0,C 180,E1 -23115.166,E2 -23115.166} C_VEL
LIN {X 0,Y 164.11,Z 694.416,A -85,B 0,C 180,E1 -23116.692,E2 -23116.692} C_VEL
LIN {X 0,Y 162.797,Z 697.093,A -85,B 0,C 180,E1 -23120.056,E2 -23120.056} C_VEL
LIN {X 0,Y 162.22,Z 698.512,A -85,B 0,C 180,E1 -23122.532,E2 -23122.532} C_VEL
LIN {X 0,Y 161.851,Z 700.053,A -85,B 0,C 180,E1 -23127.105,E2 -23127.105} C_VEL
LIN {X 0,Y 161.942,Z 700.35,A -85,B 0,C 180,E1 -23130,E2 -23130} C_VEL
LIN {X 0,Y 161.829,Z 700.069,A -85,B 0,C 180,E1 -23132.741,E2 -23132.741} C_VEL
LIN {X 0,Y 162.027,Z 698.474,A -85,B 0,C 180,E1 -23137.477,E2 -23137.477} C_VEL
LIN {X 0,Y 162.434,Z 697.032,A -85,B 0,C 180,E1 -23139.966,E2 -23139.966} C_VEL
LIN {X 0,Y 163.452,Z 694.045,A -85,B 0,C 180,E1 -23143.679,E2 -23143.679} C_VEL
LIN {X 0,Y 165.048,Z 689.998,A -85,B 0,C 180,E1 -23147.342,E2 -23147.342} C_VEL
LIN {X 0,Y 167.809,Z 683.771,A -85,B 0,C 180,E1 -23151.497,E2 -23151.497} C_VEL
LIN {X 0,Y 170.8,Z 677.003,A -85,B 0,C 180,E1 -23154.935,E2 -23154.935} C_VEL
LIN {X 0,Y 174.086,Z 669.555,A -85,B 0,C 180,E1 -23157.99,E2 -23157.99} C_VEL
LIN {X 0,Y 178.222,Z 668.23,A -85,B 0,C 180,E1 -23160.84,E2 -23160.84} C_VEL
LIN {X 0,Y 185.438,Z 665.266,A -85,B 0,C 180,E1 -23164.645,E2 -23164.645} C_VEL
LIN {X 0,Y 193.847,Z 661.038,A -85,B 0,C 180,E1 -23168.05,E2 -23168.05} C_VEL
LIN {X 0,Y 203.358,Z 655.435,A -85,B 0,C 180,E1 -23171.044,E2 -23171.044} C_VEL
LIN {X 0,Y 214.085,Z 648.086,A -85,B 0,C 180,E1 -23173.762,E2 -23173.762} C_VEL
LIN {X 0,Y 223.538,Z 640.695,A -85,B 0,C 180,E1 -23175.665,E2 -23175.665} C_VEL
LIN {X 0,Y 230.963,Z 634.187,A -85,B 0,C 180,E1 -23176.912,E2 -23176.912} C_VEL
LIN {X 0,Y 231.786,Z 633.346,A -85,B 0,C 180,E1 -23177.287,E2 -23177.287} C_VEL
LIN {X 0,Y 221.818,Z 640.445,A -85,B 0,C 180,E1 -23179.501,E2 -23179.501} C_VEL
LIN {X 0,Y 214.265,Z 644.944,A -85,B 0,C 180,E1 -23181.449,E2 -23181.449} C_VEL
LIN {X 0,Y 204.805,Z 649.52,A -85,B 0,C 180,E1 -23184.312,E2 -23184.312} C_VEL
LIN {X 0,Y 196.041,Z 652.539,A -85,B 0,C 180,E1 -23187.47,E2 -23187.47} C_VEL
LIN {X 0,Y 188.078,Z 654.153,A -85,B 0,C 180,E1 -23190.937,E2 -23190.937} C_VEL
LIN {X 0,Y 180.973,Z 654.383,A -85,B 0,C 180,E1 -23194.711,E2 -23194.711} C_VEL
LIN {X 0,Y 174.96,Z 653.155,A -85,B 0,C 180,E1 -23198.806,E2 -23198.806} C_VEL
LIN {X 0,Y 170.165,Z 650.523,A -85,B 0,C 180,E1 -23203.196,E2 -23203.196} C_VEL
LIN {X 0,Y 166.702,Z 646.454,A -85,B 0,C 180,E1 -23207.831,E2 -23207.831} C_VEL
LIN {X 0,Y 164.349,Z 640.776,A -85,B 0,C 180,E1 -23212.629,E2 -23212.629} C_VEL
LIN {X 0,Y 163.202,Z 634.382,A -85,B 0,C 180,E1 -23216.914,E2 -23216.914} C_VEL
LIN {X 0,Y 163.007,Z 626.409,A -85,B 0,C 180,E1 -23221.235,E2 -23221.235} C_VEL
LIN {X 0,Y 163.381,Z 617.995,A -85,B 0,C 180,E1 -23224.936,E2 -23224.936} C_VEL
LIN {X 0,Y 163.833,Z 608.092,A -85,B 0,C 180,E1 -23228.512,E2 -23228.512} C_VEL
LIN {X 0,Y 164.728,Z 596.176,A -85,B 0,C 180,E1 -23232.004,E2 -23232.004} C_VEL
LIN {X 0,Y 165.63,Z 584.478,A -85,B 0,C 180,E1 -23234.75,E2 -23234.75} C_VEL
LIN {X 0,Y 166.648,Z 571.586,A -85,B 0,C 180,E1 -23237.17,E2 -23237.17} C_VEL
LIN {X 0,Y 167.621,Z 559.589,A -85,B 0,C 180,E1 -23238.962,E2 -23238.962} C_VEL
LIN {X 0,Y 168.494,Z 544.207,A -85,B 0,C 180,E1 -23240.686,E2 -23240.686} C_VEL
LIN {X 0,Y 171.486,Z 480.163,A -85,B 0,C 180,E1 -23245.737,E2 -23245.737} C_VEL
LIN {X 0,Y 166.567,Z 461.76,A -85,B 0,C 180,E1 -23247.326,E2 -23247.326} C_VEL
LIN {X 0,Y 167.16,Z 462.275,A -85,B 0,C 180,E1 -23248.004,E2 -23248.004} C_VEL
LIN {X 0,Y 168.847,Z 462.294,A -85,B 0,C 180,E1 -23249.061,E2 -23249.061} C_VEL
LIN {X 0,Y 170.096,Z 464.819,A -85,B 0,C 180,E1 -23251.096,E2 -23251.096} C_VEL
LIN {X 0,Y 173.57,Z 473.324,A -85,B 0,C 180,E1 -23256.672,E2 -23256.672} C_VEL
LIN {X 0,Y 175.102,Z 477.237,A -85,B 0,C 180,E1 -23258.808,E2 -23258.808} C_VEL
LIN {X 0,Y 181.253,Z 486.887,A -85,B 0,C 180,E1 -23261.741,E2 -23261.741} C_VEL
LIN {X 0,Y 186.594,Z 496.492,A -85,B 0,C 180,E1 -23264.078,E2 -23264.078} C_VEL
LIN {X 0,Y 191.418,Z 506.157,A -85,B 0,C 180,E1 -23266.052,E2 -23266.052} C_VEL
LIN {X 0,Y 196.163,Z 517.453,A -85,B 0,C 180,E1 -23267.928,E2 -23267.928} C_VEL
LIN {X 0,Y 196.777,Z 519.9,A -85,B 0,C 180,E1 -23268.208,E2 -23268.208} C_VEL
LIN {X 0,Y 197.234,Z 524.94,A -85,B 0,C 180,E1 -23268.568,E2 -23268.568} C_VEL
LIN {X 0,Y 193.542,Z 587.65,A -85,B 0,C 180,E1 -23270.673,E2 -23270.673} C_VEL
LIN {X 0,Y 191.982,Z 601.214,A -85,B 0,C 180,E1 -23271.442,E2 -23271.442} C_VEL
LIN {X 0,Y 189.886,Z 613.38,A -85,B 0,C 180,E1 -23272.527,E2 -23272.527} C_VEL
LIN {X 0,Y 187.131,Z 625.752,A -85,B 0,C 180,E1 -23274.068,E2 -23274.068} C_VEL
LIN {X 0,Y 184.248,Z 636.117,A -85,B 0,C 180,E1 -23275.762,E2 -23275.762} C_VEL
LIN {X 0,Y 180.75,Z 646.728,A -85,B 0,C 180,E1 -23278.01,E2 -23278.01} C_VEL
LIN {X 0,Y 177.634,Z 655.394,A -85,B 0,C 180,E1 -23280.361,E2 -23280.361} C_VEL
LIN {X 0,Y 173.878,Z 664.806,A -85,B 0,C 180,E1 -23283.601,E2 -23283.601} C_VEL
LIN {X 0,Y 170.518,Z 672.278,A -85,B 0,C 180,E1 -23286.949,E2 -23286.949} C_VEL
LIN {X 0,Y 167.689,Z 678.269,A -85,B 0,C 180,E1 -23290.41,E2 -23290.41} C_VEL
LIN {X 0,Y 165.496,Z 683.002,A -85,B 0,C 180,E1 -23293.976,E2 -23293.976} C_VEL
LIN {X 0,Y 163.872,Z 686.618,A -85,B 0,C 180,E1 -23297.617,E2 -23297.617} C_VEL
LIN {X 0,Y 163.083,Z 688.478,A -85,B 0,C 180,E1 -23300.074,E2 -23300.074} C_VEL
LIN {X 0,Y 162.547,Z 689.892,A -85,B 0,C 180,E1 -23302.547,E2 -23302.547} C_VEL
LIN {X 0,Y 161.928,Z 691.495,A -85,B 0,C 180,E1 -23307.512,E2 -23307.512} C_VEL
LIN {X 0,Y 161.925,Z 691.724,A -85,B 0,C 180,E1 -23310,E2 -23310} C_VEL
LIN {X 0,Y 162.001,Z 691.279,A -85,B 0,C 180,E1 -23313.799,E2 -23313.799} C_VEL
LIN {X 0,Y 162.547,Z 689.964,A -85,B 0,C 180,E1 -23317.453,E2 -23317.453} C_VEL
LIN {X 0,Y 163.075,Z 688.591,A -85,B 0,C 180,E1 -23319.927,E2 -23319.927} C_VEL
LIN {X 0,Y 164.327,Z 685.705,A -85,B 0,C 180,E1 -23323.605,E2 -23323.605} C_VEL
LIN {X 0,Y 166.148,Z 681.779,A -85,B 0,C 180,E1 -23327.223,E2 -23327.223} C_VEL
LIN {X 0,Y 168.533,Z 676.688,A -85,B 0,C 180,E1 -23330.76,E2 -23330.76} C_VEL
LIN {X 0,Y 171.539,Z 670.266,A -85,B 0,C 180,E1 -23334.186,E2 -23334.186} C_VEL
LIN {X 0,Y 174.912,Z 662.496,A -85,B 0,C 180,E1 -23337.426,E2 -23337.426} C_VEL
LIN {X 0,Y 178.478,Z 653.297,A -85,B 0,C 180,E1 -23340.431,E2 -23340.431} C_VEL
LIN {X 0,Y 182.201,Z 642.892,A -85,B 0,C 180,E1 -23343.014,E2 -23343.014} C_VEL
LIN {X 0,Y 185.414,Z 632.691,A -85,B 0,C 180,E1 -23344.981,E2 -23344.981} C_VEL
LIN {X 0,Y 188.3,Z 621.477,A -85,B 0,C 180,E1 -23346.668,E2 -23346.668} C_VEL
LIN {X 0,Y 190.97,Z 608.726,A -85,B 0,C 180,E1 -23348.056,E2 -23348.056} C_VEL
LIN {X 0,Y 192.582,Z 597.543,A -85,B 0,C 180,E1 -23348.954,E2 -23348.954} C_VEL
LIN {X 0,Y 193.84,Z 585.458,A -85,B 0,C 180,E1 -23349.567,E2 -23349.567} C_VEL
LIN {X 0,Y 197.368,Z 524.377,A -85,B 0,C 180,E1 -23351.601,E2 -23351.601} C_VEL
LIN {X 0,Y 196.476,Z 517.979,A -85,B 0,C 180,E1 -23352.142,E2 -23352.142} C_VEL
LIN {X 0,Y 190.93,Z 504.884,A -85,B 0,C 180,E1 -23354.342,E2 -23354.342} C_VEL
LIN {X 0,Y 185.383,Z 494.039,A -85,B 0,C 180,E1 -23356.643,E2 -23356.643} C_VEL
LIN {X 0,Y 179.962,Z 484.841,A -85,B 0,C 180,E1 -23359.053,E2 -23359.053} C_VEL
LIN {X 0,Y 174.924,Z 476.827,A -85,B 0,C 180,E1 -23361.544,E2 -23361.544} C_VEL
LIN {X 0,Y 173.67,Z 473.558,A -85,B 0,C 180,E1 -23363.424,E2 -23363.424} C_VEL
LIN {X 0,Y 173.091,Z 472.654,A -85,B 0,C 180,E1 -23364.076,E2 -23364.076} C_VEL
LIN {X 0,Y 168.24,Z 470.271,A -85,B 0,C 180,E1 -23367.643,E2 -23367.643} C_VEL
LIN {X 0,Y 167.915,Z 469.573,A -85,B 0,C 180,E1 -23368.179,E2 -23368.179} C_VEL
LIN {X 0,Y 169.523,Z 477.346,A -85,B 0,C 180,E1 -23370.721,E2 -23370.721} C_VEL
LIN {X 0,Y 171.441,Z 505.634,A -85,B 0,C 180,E1 -23372.944,E2 -23372.944} C_VEL
LIN {X 0,Y 172.191,Z 513.582,A -85,B 0,C 180,E1 -23373.564,E2 -23373.564} C_VEL
LIN {X 0,Y 168.506,Z 586.307,A -85,B 0,C 180,E1 -23379.236,E2 -23379.236} C_VEL
LIN {X 0,Y 167.684,Z 600.776,A -85,B 0,C 180,E1 -23380.728,E2 -23380.728} C_VEL
LIN {X 0,Y 166.586,Z 615.4,A -85,B 0,C 180,E1 -23382.823,E2 -23382.823} C_VEL
LIN {X 0,Y 165.579,Z 628.319,A -85,B 0,C 180,E1 -23385.246,E2 -23385.246} C_VEL
LIN {X 0,Y 164.633,Z 639.945,A -85,B 0,C 180,E1 -23387.988,E2 -23387.988} C_VEL
LIN {X 0,Y 163.843,Z 650.417,A -85,B 0,C 180,E1 -23391.034,E2 -23391.034} C_VEL
LIN {X 0,Y 163.41,Z 658.309,A -85,B 0,C 180,E1 -23393.827,E2 -23393.827} C_VEL
LIN {X 0,Y 163.049,Z 666.919,A -85,B 0,C 180,E1 -23397.529,E2 -23397.529} C_VEL
LIN {X 0,Y 162.903,Z 673.93,A -85,B 0,C 180,E1 -23401.236,E2 -23401.236} C_VEL
LIN {X 0,Y 162.886,Z 679.478,A -85,B 0,C 180,E1 -23404.95,E2 -23404.95} C_VEL
LIN {X 0,Y 163.332,Z 683.847,A -85,B 0,C 180,E1 -23408.537,E2 -23408.537} C_VEL
LIN {X 0,Y 164.5,Z 687.543,A -85,B 0,C 180,E1 -23412.334,E2 -23412.334} C_VEL
LIN {X 0,Y 167.215,Z 691.026,A -85,B 0,C 180,E1 -23417.11,E2 -23417.11} C_VEL
LIN {X 0,Y 171.212,Z 693.103,A -85,B 0,C 180,E1 -23421.681,E2 -23421.681} C_VEL
LIN {X 0,Y 173.689,Z 693.633,A -85,B 0,C 180,E1 -23423.868,E2 -23423.868} C_VEL
LIN {X 0,Y 179.824,Z 693.694,A -85,B 0,C 180,E1 -23427.969,E2 -23427.969} C_VEL
LIN {X 0,Y 187.027,Z 692.427,A -85,B 0,C 180,E1 -23431.741,E2 -23431.741} C_VEL
LIN {X 0,Y 195.242,Z 689.75,A -85,B 0,C 180,E1 -23435.166,E2 -23435.166} C_VEL
LIN {X 0,Y 204.221,Z 685.727,A -85,B 0,C 180,E1 -23438.177,E2 -23438.177} C_VEL
LIN {X 0,Y 206.351,Z 684.612,A -85,B 0,C 180,E1 -23439.071,E2 -23439.071} C_VEL
LIN {X 0,Y 211.242,Z 681.645,A -85,B 0,C 180,E1 -23442.427,E2 -23442.427} C_VEL
LIN {X 0,Y 213.579,Z 680.241,A -85,B 0,C 180,E1 -23443.204,E2 -23443.204} C_VEL
LIN {X 0,Y 217.881,Z 677.594,A -85,B 0,C 180,E1 -23444.121,E2 -23444.121} C_VEL
LIN {X 0,Y 217.554,Z 677.874,A -85,B 0,C 180,E1 -23444.708,E2 -23444.708} C_VEL
LIN {X 0,Y 209.157,Z 683.257,A -85,B 0,C 180,E1 -23446.462,E2 -23446.462} C_VEL
LIN {X 0,Y 198.696,Z 688.945,A -85,B 0,C 180,E1 -23449.129,E2 -23449.129} C_VEL
LIN {X 0,Y 191.369,Z 692.267,A -85,B 0,C 180,E1 -23451.367,E2 -23451.367} C_VEL
LIN {X 0,Y 182.477,Z 695.424,A -85,B 0,C 180,E1 -23454.71,E2 -23454.71} C_VEL
LIN {X 0,Y 174.587,Z 697.281,A -85,B 0,C 180,E1 -23458.445,E2 -23458.445} C_VEL
LIN {X 0,Y 167.973,Z 697.881,A -85,B 0,C 180,E1 -23462.597,E2 -23462.597} C_VEL
LIN {X 0,Y 162.901,Z 697.252,A -85,B 0,C 180,E1 -23467.152,E2 -23467.152} C_VEL
LIN {X 0,Y 160.77,Z 696.463,A -85,B 0,C 180,E1 -23469.53,E2 -23469.53} C_VEL
LIN {X 0,Y 157.965,Z 693.932,A -85,B 0,C 180,E1 -23474.517,E2 -23474.517} C_VEL
LIN {X 0,Y 157.637,Z 693.49,A -85,B 0,C 180,E1 -23475.311,E2 -23475.311} C_VEL
LIN {X 0,Y 155.812,Z 696.905,A -85,B 0,C 180,E1 -23479.606,E2 -23479.606} C_VEL
LIN {X 0,Y 155.187,Z 698.323,A -85,B 0,C 180,E1 -23482.191,E2 -23482.191} C_VEL
LIN {X 0,Y 154.776,Z 699.944,A -85,B 0,C 180,E1 -23487.397,E2 -23487.397} C_VEL
LIN {X 0,Y 154.853,Z 700.161,A -85,B 0,C 180,E1 -23490,E2 -23490} C_VEL
LIN {X 0,Y 154.739,Z 699.929,A -85,B 0,C 180,E1 -23492.603,E2 -23492.603} C_VEL
LIN {X 0,Y 154.761,Z 699.302,A -85,B 0,C 180,E1 -23495.211,E2 -23495.211} C_VEL
LIN {X 0,Y 154.972,Z 698.285,A -85,B 0,C 180,E1 -23497.819,E2 -23497.819} C_VEL
LIN {X 0,Y 155.431,Z 696.843,A -85,B 0,C 180,E1 -23500.42,E2 -23500.42} C_VEL
LIN {X 0,Y 156.524,Z 693.855,A -85,B 0,C 180,E1 -23504.297,E2 -23504.297} C_VEL
LIN {X 0,Y 158.274,Z 689.808,A -85,B 0,C 180,E1 -23508.109,E2 -23508.109} C_VEL
LIN {X 0,Y 161.184,Z 683.581,A -85,B 0,C 180,E1 -23512.428,E2 -23512.428} C_VEL
LIN {X 0,Y 163.82,Z 678.019,A -85,B 0,C 180,E1 -23515.405,E2 -23515.405} C_VEL
LIN {X 0,Y 166.784,Z 671.328,A -85,B 0,C 180,E1 -23518.298,E2 -23518.298} C_VEL
LIN {X 0,Y 168.054,Z 668.822,A -85,B 0,C 180,E1 -23519.26,E2 -23519.26} C_VEL
LIN {X 0,Y 172.169,Z 667.82,A -85,B 0,C 180,E1 -23522.051,E2 -23522.051} C_VEL
LIN {X 0,Y 179.644,Z 665.337,A -85,B 0,C 180,E1 -23525.932,E2 -23525.932} C_VEL
LIN {X 0,Y 188.323,Z 661.653,A -85,B 0,C 180,E1 -23529.377,E2 -23529.377} C_VEL
LIN {X 0,Y 198.094,Z 656.682,A -85,B 0,C 180,E1 -23532.383,E2 -23532.383} C_VEL
LIN {X 0,Y 208.889,Z 650.186,A -85,B 0,C 180,E1 -23535.046,E2 -23535.046} C_VEL
LIN {X 0,Y 218.729,Z 643.392,A -85,B 0,C 180,E1 -23536.969,E2 -23536.969} C_VEL
LIN {X 0,Y 220.197,Z 642.286,A -85,B 0,C 180,E1 -23537.23,E2 -23537.23} C_VEL
LIN {X 0,Y 219.622,Z 642.474,A -85,B 0,C 180,E1 -23537.778,E2 -23537.778} C_VEL
LIN {X 0,Y 211.95,Z 646.644,A -85,B 0,C 180,E1 -23539.59,E2 -23539.59} C_VEL
LIN {X 0,Y 204.18,Z 650.131,A -85,B 0,C 180,E1 -23541.715,E2 -23541.715} C_VEL
LIN {X 0,Y 194.71,Z 653.362,A -85,B 0,C 180,E1 -23544.724,E2 -23544.724} C_VEL
LIN {X 0,Y 186.033,Z 655.12,A -85,B 0,C 180,E1 -23548.069,E2 -23548.069} C_VEL
LIN {X 0,Y 178.189,Z 655.529,A -85,B 0,C 180,E1 -23551.752,E2 -23551.752} C_VEL
LIN {X 0,Y 171.353,Z 654.569,A -85,B 0,C 180,E1 -23555.786,E2 -23555.786} C_VEL
LIN {X 0,Y 165.695,Z 652.173,A -85,B 0,C 180,E1 -23560.164,E2 -23560.164} C_VEL
LIN {X 0,Y 161.442,Z 648.373,A -85,B 0,C 180,E1 -23564.859,E2 -23564.859} C_VEL
LIN {X 0,Y 158.427,Z 643.104,A -85,B 0,C 180,E1 -23569.779,E2 -23569.779} C_VEL
LIN {X 0,Y 156.6,Z 636.093,A -85,B 0,C 180,E1 -23574.85,E2 -23574.85} C_VEL
LIN {X 0,Y 156.034,Z 628.419,A -85,B 0,C 180,E1 -23579.355,E2 -23579.355} C_VEL
LIN {X 0,Y 156.293,Z 620.384,A -85,B 0,C 180,E1 -23583.222,E2 -23583.222} C_VEL
LIN {X 0,Y 156.536,Z 612.279,A -85,B 0,C 180,E1 -23586.445,E2 -23586.445} C_VEL
LIN {X 0,Y 157.207,Z 601.534,A -85,B 0,C 180,E1 -23589.992,E2 -23589.992} C_VEL
LIN {X 0,Y 158.158,Z 589.775,A -85,B 0,C 180,E1 -23593.164,E2 -23593.164} C_VEL
LIN {X 0,Y 159.197,Z 576.601,A -85,B 0,C 180,E1 -23596.017,E2 -23596.017} C_VEL
LIN {X 0,Y 160.335,Z 562.61,A -85,B 0,C 180,E1 -23598.364,E2 -23598.364} C_VEL
LIN {X 0,Y 161.201,Z 548.167,A -85,B 0,C 180,E1 -23600.163,E2 -23600.163} C_VEL
LIN {X 0,Y 162.162,Z 526.963,A -85,B 0,C 180,E1 -23602.034,E2 -23602.034} C_VEL
LIN {X 0,Y 164.322,Z 481.04,A -85,B 0,C 180,E1 -23605.798,E2 -23605.798} C_VEL
LIN {X 0,Y 160.837,Z 468.057,A -85,B 0,C 180,E1 -23606.972,E2 -23606.972} C_VEL
LIN {X 0,Y 161.244,Z 468.568,A -85,B 0,C 180,E1 -23607.552,E2 -23607.552} C_VEL
LIN {X 0,Y 162.535,Z 468.52,A -85,B 0,C 180,E1 -23608.401,E2 -23608.401} C_VEL
LIN {X 0,Y 165.151,Z 469.789,A -85,B 0,C 180,E1 -23610.708,E2 -23610.708} C_VEL
LIN {X 0,Y 168.112,Z 477.215,A -85,B 0,C 180,E1 -23615.73,E2 -23615.73} C_VEL
LIN {X 0,Y 174.999,Z 487.715,A -85,B 0,C 180,E1 -23619.437,E2 -23619.437} C_VEL
LIN {X 0,Y 180.859,Z 497.924,A -85,B 0,C 180,E1 -23622.246,E2 -23622.246} C_VEL
LIN {X 0,Y 186.175,Z 508.503,A -85,B 0,C 180,E1 -23624.597,E2 -23624.597} C_VEL
LIN {X 0,Y 191.179,Z 520.532,A -85,B 0,C 180,E1 -23626.717,E2 -23626.717} C_VEL
LIN {X 0,Y 191.617,Z 522.297,A -85,B 0,C 180,E1 -23626.93,E2 -23626.93} C_VEL
LIN {X 0,Y 191.897,Z 526.133,A -85,B 0,C 180,E1 -23627.201,E2 -23627.201} C_VEL
LIN {X 0,Y 188.121,Z 587.515,A -85,B 0,C 180,E1 -23629.29,E2 -23629.29} C_VEL
LIN {X 0,Y 186.612,Z 600.733,A -85,B 0,C 180,E1 -23630.047,E2 -23630.047} C_VEL
LIN {X 0,Y 184.539,Z 612.47,A -85,B 0,C 180,E1 -23631.069,E2 -23631.069} C_VEL
LIN {X 0,Y 181.873,Z 624.223,A -85,B 0,C 180,E1 -23632.51,E2 -23632.51} C_VEL
LIN {X 0,Y 178.872,Z 634.915,A -85,B 0,C 180,E1 -23634.236,E2 -23634.236} C_VEL
LIN {X 0,Y 175.146,Z 645.869,A -85,B 0,C 180,E1 -23636.513,E2 -23636.513} C_VEL
LIN {X 0,Y 171.502,Z 655.58,A -85,B 0,C 180,E1 -23639.188,E2 -23639.188} C_VEL
LIN {X 0,Y 168.16,Z 663.662,A -85,B 0,C 180,E1 -23642.01,E2 -23642.01} C_VEL
LIN {X 0,Y 164.546,Z 671.35,A -85,B 0,C 180,E1 -23645.39,E2 -23645.39} C_VEL
LIN {X 0,Y 161.941,Z 676.619,A -85,B 0,C 180,E1 -23648.353,E2 -23648.353} C_VEL
LIN {X 0,Y 159.419,Z 681.762,A -85,B 0,C 180,E1 -23652.025,E2 -23652.025} C_VEL
LIN {X 0,Y 157.44,Z 685.74,A -85,B 0,C 180,E1 -23655.788,E2 -23655.788} C_VEL
LIN {X 0,Y 156.084,Z 688.667,A -85,B 0,C 180,E1 -23659.624,E2 -23659.624} C_VEL
LIN {X 0,Y 155.506,Z 690.082,A -85,B 0,C 180,E1 -23662.208,E2 -23662.208} C_VEL
LIN {X 0,Y 154.845,Z 691.684,A -85,B 0,C 180,E1 -23667.399,E2 -23667.399} C_VEL
LIN {X 0,Y 154.827,Z 691.913,A -85,B 0,C 180,E1 -23670,E2 -23670} C_VEL
LIN {X 0,Y 154.859,Z 691.607,A -85,B 0,C 180,E1 -23673.205,E2 -23673.205} C_VEL
LIN {X 0,Y 155.505,Z 690.153,A -85,B 0,C 180,E1 -23677.792,E2 -23677.792} C_VEL
LIN {X 0,Y 156.077,Z 688.779,A -85,B 0,C 180,E1 -23680.377,E2 -23680.377} C_VEL
LIN {X 0,Y 157.426,Z 685.893,A -85,B 0,C 180,E1 -23684.214,E2 -23684.214} C_VEL
LIN {X 0,Y 159.388,Z 681.966,A -85,B 0,C 180,E1 -23687.978,E2 -23687.978} C_VEL
LIN {X 0,Y 161.918,Z 676.873,A -85,B 0,C 180,E1 -23691.65,E2 -23691.65} C_VEL
LIN {X 0,Y 165.098,Z 670.45,A -85,B 0,C 180,E1 -23695.194,E2 -23695.194} C_VEL
LIN {X 0,Y 168.498,Z 662.962,A -85,B 0,C 180,E1 -23698.431,E2 -23698.431} C_VEL
LIN {X 0,Y 172.007,Z 654.471,A -85,B 0,C 180,E1 -23701.328,E2 -23701.328} C_VEL
LIN {X 0,Y 175.512,Z 645.351,A -85,B 0,C 180,E1 -23703.752,E2 -23703.752} C_VEL
LIN {X 0,Y 179.233,Z 634.246,A -85,B 0,C 180,E1 -23706.028,E2 -23706.028} C_VEL
LIN {X 0,Y 182.205,Z 623.399,A -85,B 0,C 180,E1 -23707.758,E2 -23707.758} C_VEL
LIN {X 0,Y 185.001,Z 611.349,A -85,B 0,C 180,E1 -23709.166,E2 -23709.166} C_VEL
LIN {X 0,Y 186.872,Z 599.42,A -85,B 0,C 180,E1 -23710.203,E2 -23710.203} C_VEL
LIN {X 0,Y 188.344,Z 586.563,A -85,B 0,C 180,E1 -23710.895,E2 -23710.895} C_VEL
LIN {X 0,Y 192.029,Z 525.134,A -85,B 0,C 180,E1 -23712.996,E2 -23712.996} C_VEL
LIN {X 0,Y 191.495,Z 521.016,A -85,B 0,C 180,E1 -23713.353,E2 -23713.353} C_VEL
LIN {X 0,Y 185.967,Z 507.838,A -85,B 0,C 180,E1 -23715.697,E2 -23715.697} C_VEL
LIN {X 0,Y 180.166,Z 496.541,A -85,B 0,C 180,E1 -23718.285,E2 -23718.285} C_VEL
LIN {X 0,Y 174.234,Z 486.517,A -85,B 0,C 180,E1 -23721.17,E2 -23721.17} C_VEL
LIN {X 0,Y 170.314,Z 480.61,A -85,B 0,C 180,E1 -23723.249,E2 -23723.249} C_VEL
LIN {X 0,Y 168.485,Z 478.134,A -85,B 0,C 180,E1 -23724.269,E2 -23724.269} C_VEL
LIN {X 0,Y 166.619,Z 477.094,A -85,B 0,C 180,E1 -23725.289,E2 -23725.289} C_VEL
LIN {X 0,Y 162.115,Z 475.173,A -85,B 0,C 180,E1 -23728.652,E2 -23728.652} C_VEL
LIN {X 0,Y 161.672,Z 474.375,A -85,B 0,C 180,E1 -23729.402,E2 -23729.402} C_VEL
LIN {X 0,Y 162.403,Z 477.805,A -85,B 0,C 180,E1 -23730.473,E2 -23730.473} C_VEL
LIN {X 0,Y 164.583,Z 508.018,A -85,B 0,C 180,E1 -23732.958,E2 -23732.958} C_VEL
LIN {X 0,Y 165.063,Z 514.256,A -85,B 0,C 180,E1 -23733.466,E2 -23733.466} C_VEL
LIN {X 0,Y 161.442,Z 585.716,A -85,B 0,C 180,E1 -23739.369,E2 -23739.369} C_VEL
LIN {X 0,Y 160.661,Z 599.708,A -85,B 0,C 180,E1 -23740.847,E2 -23740.847} C_VEL
LIN {X 0,Y 159.7,Z 612.703,A -85,B 0,C 180,E1 -23742.719,E2 -23742.719} C_VEL
LIN {X 0,Y 158.801,Z 624.758,A -85,B 0,C 180,E1 -23744.929,E2 -23744.929} C_VEL
LIN {X 0,Y 157.81,Z 636.908,A -85,B 0,C 180,E1 -23747.788,E2 -23747.788} C_VEL
LIN {X 0,Y 157.072,Z 647.2,A -85,B 0,C 180,E1 -23750.757,E2 -23750.757} C_VEL
LIN {X 0,Y 156.541,Z 656.956,A -85,B 0,C 180,E1 -23754.202,E2 -23754.202} C_VEL
LIN {X 0,Y 156.163,Z 665.857,A -85,B 0,C 180,E1 -23758.066,E2 -23758.066} C_VEL
LIN {X 0,Y 156.039,Z 672.926,A -85,B 0,C 180,E1 -23761.936,E2 -23761.936} C_VEL
LIN {X 0,Y 156.009,Z 677.804,A -85,B 0,C 180,E1 -23765.169,E2 -23765.169} C_VEL
LIN {X 0,Y 156.381,Z 682.111,A -85,B 0,C 180,E1 -23768.614,E2 -23768.614} C_VEL
LIN {X 0,Y 157.675,Z 686.473,A -85,B 0,C 180,E1 -23772.877,E2 -23772.877} C_VEL
LIN {X 0,Y 160.472,Z 690.362,A -85,B 0,C 180,E1 -23777.853,E2 -23777.853} C_VEL
LIN {X 0,Y 164.636,Z 692.853,A -85,B 0,C 180,E1 -23782.594,E2 -23782.594} C_VEL
LIN {X 0,Y 170.307,Z 694.044,A -85,B 0,C 180,E1 -23786.996,E2 -23786.996} C_VEL
LIN {X 0,Y 177.233,Z 693.94,A -85,B 0,C 180,E1 -23791.031,E2 -23791.031} C_VEL
LIN {X 0,Y 185.211,Z 692.481,A -85,B 0,C 180,E1 -23794.694,E2 -23794.694} C_VEL
LIN {X 0,Y 194.226,Z 689.67,A -85,B 0,C 180,E1 -23797.962,E2 -23797.962} C_VEL
LIN {X 0,Y 204.107,Z 685.438,A -85,B 0,C 180,E1 -23800.861,E2 -23800.861} C_VEL
LIN {X 0,Y 213.579,Z 680.241,A -85,B 0,C 180,E1 -23803.204,E2 -23803.204} C_VEL
LIN {X 0,Y 212.261,Z 681.06,A -85,B 0,C 180,E1 -23803.283,E2 -23803.283} C_VEL
LIN {X 0,Y 207.502,Z 683.666,A -85,B 0,C 180,E1 -23802.855,E2 -23802.855} C_VEL
LIN {X 0,Y 201.461,Z 686.571,A -85,B 0,C 180,E1 -23801.962,E2 -23801.962} C_VEL
LIN {X 0,Y 196.785,Z 688.537,A -85,B 0,C 180,E1 -23801.153,E2 -23801.153} C_VEL
LIN {X 0,Y 190.177,Z 690.885,A -85,B 0,C 180,E1 -23799.655,E2 -23799.655} C_VEL
LIN {X 0,Y 188.167,Z 691.451,A -85,B 0,C 180,E1 -23799.054,E2 -23799.054} C_VEL
LIN {X 0,Y 179.486,Z 693.536,A -85,B 0,C 180,E1 -23795.969,E2 -23795.969} C_VEL
LIN {X 0,Y 171.206,Z 694.473,A -85,B 0,C 180,E1 -23792.252,E2 -23792.252} C_VEL
LIN {X 0,Y 164.023,Z 694.098,A -85,B 0,C 180,E1 -23788.12,E2 -23788.12} C_VEL
LIN {X 0,Y 158.115,Z 692.426,A -85,B 0,C 180,E1 -23783.581,E2 -23783.581} C_VEL
LIN {X 0,Y 153.79,Z 689.504,A -85,B 0,C 180,E1 -23778.656,E2 -23778.656} C_VEL
LIN {X 0,Y 150.886,Z 685.251,A -85,B 0,C 180,E1 -23773.467,E2 -23773.467} C_VEL
LIN {X 0,Y 149.409,Z 679.404,A -85,B 0,C 180,E1 -23768.112,E2 -23768.112} C_VEL
LIN {X 0,Y 149.209,Z 672.942,A -85,B 0,C 180,E1 -23763.375,E2 -23763.375} C_VEL
LIN {X 0,Y 149.344,Z 665.898,A -85,B 0,C 180,E1 -23759.326,E2 -23759.326} C_VEL
LIN {X 0,Y 149.577,Z 657.129,A -85,B 0,C 180,E1 -23755.283,E2 -23755.283} C_VEL
LIN {X 0,Y 149.958,Z 650.194,A -85,B 0,C 180,E1 -23752.595,E2 -23752.595} C_VEL
LIN {X 0,Y 150.691,Z 638.537,A -85,B 0,C 180,E1 -23748.908,E2 -23748.908} C_VEL
LIN {X 0,Y 151.609,Z 626.695,A -85,B 0,C 180,E1 -23745.914,E2 -23745.914} C_VEL
LIN {X 0,Y 152.591,Z 613.489,A -85,B 0,C 180,E1 -23743.27,E2 -23743.27} C_VEL
LIN {X 0,Y 153.562,Z 599.663,A -85,B 0,C 180,E1 -23741.142,E2 -23741.142} C_VEL
LIN {X 0,Y 154.453,Z 584.325,A -85,B 0,C 180,E1 -23739.438,E2 -23739.438} C_VEL
LIN {X 0,Y 157.925,Z 512.073,A -85,B 0,C 180,E1 -23733.177,E2 -23733.177} C_VEL
LIN {X 0,Y 155.743,Z 485.011,A -85,B 0,C 180,E1 -23730.793,E2 -23730.793} C_VEL
LIN {X 0,Y 156.243,Z 487.038,A -85,B 0,C 180,E1 -23730.281,E2 -23730.281} C_VEL
LIN {X 0,Y 157.36,Z 487.036,A -85,B 0,C 180,E1 -23729.575,E2 -23729.575} C_VEL
LIN {X 0,Y 158.898,Z 484.546,A -85,B 0,C 180,E1 -23728.854,E2 -23728.854} C_VEL
LIN {X 0,Y 160.065,Z 482.009,A -85,B 0,C 180,E1 -23728.381,E2 -23728.381} C_VEL
LIN {X 0,Y 166.123,Z 484.59,A -85,B 0,C 180,E1 -23724.938,E2 -23724.938} C_VEL
LIN {X 0,Y 170.056,Z 490.64,A -85,B 0,C 180,E1 -23722.673,E2 -23722.673} C_VEL
LIN {X 0,Y 175.969,Z 500.641,A -85,B 0,C 180,E1 -23719.591,E2 -23719.591} C_VEL
LIN {X 0,Y 181.835,Z 512.451,A -85,B 0,C 180,E1 -23716.788,E2 -23716.788} C_VEL
LIN {X 0,Y 186.643,Z 524.184,A -85,B 0,C 180,E1 -23714.61,E2 -23714.61} C_VEL
LIN {X 0,Y 186.843,Z 527.326,A -85,B 0,C 180,E1 -23714.383,E2 -23714.383} C_VEL
LIN {X 0,Y 182.849,Z 588.799,A -85,B 0,C 180,E1 -23712.256,E2 -23712.256} C_VEL
LIN {X 0,Y 181.163,Z 601.825,A -85,B 0,C 180,E1 -23711.493,E2 -23711.493} C_VEL
LIN {X 0,Y 178.821,Z 614.823,A -85,B 0,C 180,E1 -23710.243,E2 -23710.243} C_VEL
LIN {X 0,Y 175.747,Z 626.974,A -85,B 0,C 180,E1 -23708.67,E2 -23708.67} C_VEL
LIN {X 0,Y 172.235,Z 638.404,A -85,B 0,C 180,E1 -23706.639,E2 -23706.639} C_VEL
LIN {X 0,Y 168.394,Z 648.68,A -85,B 0,C 180,E1 -23704.293,E2 -23704.293} C_VEL
LIN {X 0,Y 164.631,Z 657.951,A -85,B 0,C 180,E1 -23701.53,E2 -23701.53} C_VEL
LIN {X 0,Y 160.579,Z 666.854,A -85,B 0,C 180,E1 -23698.066,E2 -23698.066} C_VEL
LIN {X 0,Y 156.96,Z 674.024,A -85,B 0,C 180,E1 -23694.467,E2 -23694.467} C_VEL
LIN {X 0,Y 154.319,Z 678.875,A -85,B 0,C 180,E1 -23691.367,E2 -23691.367} C_VEL
LIN {X 0,Y 151.863,Z 683.561,A -85,B 0,C 180,E1 -23687.506,E2 -23687.506} C_VEL
LIN {X 0,Y 149.997,Z 687.13,A -85,B 0,C 180,E1 -23683.549,E2 -23683.549} C_VEL
LIN {X 0,Y 149.103,Z 688.967,A -85,B 0,C 180,E1 -23680.868,E2 -23680.868} C_VEL
LIN {X 0,Y 148.467,Z 690.341,A -85,B 0,C 180,E1 -23678.164,E2 -23678.164} C_VEL
LIN {X 0,Y 148.011,Z 691.314,A -85,B 0,C 180,E1 -23675.449,E2 -23675.449} C_VEL
LIN {X 0,Y 147.756,Z 691.904,A -85,B 0,C 180,E1 -23672.726,E2 -23672.726} C_VEL
LIN {X 0,Y 147.746,Z 692.101,A -85,B 0,C 180,E1 -23670,E2 -23670} C_VEL
LIN {X 0,Y 148.011,Z 691.263,A -85,B 0,C 180,E1 -23664.551,E2 -23664.551} C_VEL
LIN {X 0,Y 148.468,Z 690.271,A -85,B 0,C 180,E1 -23661.836,E2 -23661.836} C_VEL
LIN {X 0,Y 149.109,Z 688.857,A -85,B 0,C 180,E1 -23659.133,E2 -23659.133} C_VEL
LIN {X 0,Y 150.567,Z 685.929,A -85,B 0,C 180,E1 -23655.124,E2 -23655.124} C_VEL
LIN {X 0,Y 152.69,Z 681.951,A -85,B 0,C 180,E1 -23651.204,E2 -23651.204} C_VEL
LIN {X 0,Y 155.37,Z 676.807,A -85,B 0,C 180,E1 -23647.388,E2 -23647.388} C_VEL
LIN {X 0,Y 158.745,Z 670.331,A -85,B 0,C 180,E1 -23643.722,E2 -23643.722} C_VEL
LIN {X 0,Y 162.781,Z 661.826,A -85,B 0,C 180,E1 -23640.012,E2 -23640.012} C_VEL
LIN {X 0,Y 166.187,Z 654.01,A -85,B 0,C 180,E1 -23637.372,E2 -23637.372} C_VEL
LIN {X 0,Y 170.132,Z 643.797,A -85,B 0,C 180,E1 -23634.667,E2 -23634.667} C_VEL
LIN {X 0,Y 174.046,Z 632.326,A -85,B 0,C 180,E1 -23632.356,E2 -23632.356} C_VEL
LIN {X 0,Y 177.235,Z 620.826,A -85,B 0,C 180,E1 -23630.62,E2 -23630.62} C_VEL
LIN {X 0,Y 180.015,Z 607.77,A -85,B 0,C 180,E1 -23629.16,E2 -23629.16} C_VEL
LIN {X 0,Y 182.079,Z 594.71,A -85,B 0,C 180,E1 -23628.202,E2 -23628.202} C_VEL
LIN {X 0,Y 183.308,Z 581.476,A -85,B 0,C 180,E1 -23627.611,E2 -23627.611} C_VEL
LIN {X 0,Y 186.675,Z 525.696,A -85,B 0,C 180,E1 -23625.67,E2 -23625.67} C_VEL
LIN {X 0,Y 186.183,Z 523.325,A -85,B 0,C 180,E1 -23625.395,E2 -23625.395} C_VEL
LIN {X 0,Y 181.097,Z 510.97,A -85,B 0,C 180,E1 -23623.079,E2 -23623.079} C_VEL
LIN {X 0,Y 175.167,Z 499.379,A -85,B 0,C 180,E1 -23620.237,E2 -23620.237} C_VEL
LIN {X 0,Y 170.061,Z 490.682,A -85,B 0,C 180,E1 -23617.563,E2 -23617.563} C_VEL
LIN {X 0,Y 164.482,Z 482.044,A -85,B 0,C 180,E1 -23614.297,E2 -23614.297} C_VEL
LIN {X 0,Y 160.987,Z 476.95,A -85,B 0,C 180,E1 -23611.914,E2 -23611.914} C_VEL
LIN {X 0,Y 160.045,Z 474.988,A -85,B 0,C 180,E1 -23610.331,E2 -23610.331} C_VEL
LIN {X 0,Y 158.748,Z 474.359,A -85,B 0,C 180,E1 -23609.143,E2 -23609.143} C_VEL
LIN {X 0,Y 155.235,Z 474.552,A -85,B 0,C 180,E1 -23606.731,E2 -23606.731} C_VEL
LIN {X 0,Y 155.242,Z 474.568,A -85,B 0,C 180,E1 -23606.522,E2 -23606.522} C_VEL
LIN {X 0,Y 157.169,Z 482.056,A -85,B 0,C 180,E1 -23605.845,E2 -23605.845} C_VEL
LIN {X 0,Y 154.346,Z 543.234,A -85,B 0,C 180,E1 -23600.49,E2 -23600.49} C_VEL
LIN {X 0,Y 153.556,Z 557.221,A -85,B 0,C 180,E1 -23598.859,E2 -23598.859} C_VEL
LIN {X 0,Y 152.693,Z 568.864,A -85,B 0,C 180,E1 -23597.063,E2 -23597.063} C_VEL
LIN {X 0,Y 151.65,Z 582.411,A -85,B 0,C 180,E1 -23594.424,E2 -23594.424} C_VEL
LIN {X 0,Y 150.674,Z 595.132,A -85,B 0,C 180,E1 -23591.279,E2 -23591.279} C_VEL
LIN {X 0,Y 149.909,Z 605.639,A -85,B 0,C 180,E1 -23588.085,E2 -23588.085} C_VEL
LIN {X 0,Y 149.462,Z 616.441,A -85,B 0,C 180,E1 -23584.045,E2 -23584.045} C_VEL
LIN {X 0,Y 149.122,Z 625.223,A -85,B 0,C 180,E1 -23580,E2 -23580} C_VEL
LIN {X 0,Y 149.52,Z 633.62,A -85,B 0,C 180,E1 -23575.282,E2 -23575.282} C_VEL
LIN {X 0,Y 150.953,Z 640.457,A -85,B 0,C 180,E1 -23570.622,E2 -23570.622} C_VEL
LIN {X 0,Y 153.716,Z 646.629,A -85,B 0,C 180,E1 -23565.436,E2 -23565.436} C_VEL
LIN {X 0,Y 156.669,Z 650.211,A -85,B 0,C 180,E1 -23561.699,E2 -23561.699} C_VEL
LIN {X 0,Y 161.823,Z 653.752,A -85,B 0,C 180,E1 -23556.991,E2 -23556.991} C_VEL
LIN {X 0,Y 168.334,Z 655.891,A -85,B 0,C 180,E1 -23552.661,E2 -23552.661} C_VEL
LIN {X 0,Y 176,Z 656.672,A -85,B 0,C 180,E1 -23548.727,E2 -23548.727} C_VEL
LIN {X 0,Y 184.571,Z 656.118,A -85,B 0,C 180,E1 -23545.169,E2 -23545.169} C_VEL
LIN {X 0,Y 193.955,Z 654.184,A -85,B 0,C 180,E1 -23541.975,E2 -23541.975} C_VEL
LIN {X 0,Y 204.052,Z 650.855,A -85,B 0,C 180,E1 -23539.126,E2 -23539.126} C_VEL
LIN {X 0,Y 209.351,Z 648.649,A -85,B 0,C 180,E1 -23537.824,E2 -23537.824} C_VEL
LIN {X 0,Y 209.513,Z 648.67,A -85,B 0,C 180,E1 -23537.56,E2 -23537.56} C_VEL
LIN {X 0,Y 198.283,Z 655.047,A -85,B 0,C 180,E1 -23535.145,E2 -23535.145} C_VEL
LIN {X 0,Y 187.798,Z 660.071,A -85,B 0,C 180,E1 -23532.347,E2 -23532.347} C_VEL
LIN {X 0,Y 178.299,Z 663.812,A -85,B 0,C 180,E1 -23529.1,E2 -23529.1} C_VEL
LIN {X 0,Y 169.93,Z 666.379,A -85,B 0,C 180,E1 -23525.381,E2 -23525.381} C_VEL
LIN {X 0,Y 162.495,Z 667.89,A -85,B 0,C 180,E1 -23520.904,E2 -23520.904} C_VEL
LIN {X 0,Y 162.103,Z 668.109,A -85,B 0,C 180,E1 -23520.626,E2 -23520.626} C_VEL
LIN {X 0,Y 158.559,Z 675.267,A -85,B 0,C 180,E1 -23517.76,E2 -23517.76} C_VEL
LIN {X 0,Y 155.169,Z 682.388,A -85,B 0,C 180,E1 -23514.056,E2 -23514.056} C_VEL
LIN {X 0,Y 152.344,Z 688.01,A -85,B 0,C 180,E1 -23510.242,E2 -23510.242} C_VEL
LIN {X 0,Y 150.125,Z 692.423,A -85,B 0,C 180,E1 -23506.313,E2 -23506.313} C_VEL
LIN {X 0,Y 149.153,Z 694.752,A -85,B 0,C 180,E1 -23503.627,E2 -23503.627} C_VEL
LIN {X 0,Y 148.414,Z 696.652,A -85,B 0,C 180,E1 -23500.919,E2 -23500.919} C_VEL
LIN {X 0,Y 147.918,Z 698.095,A -85,B 0,C 180,E1 -23498.195,E2 -23498.195} C_VEL
LIN {X 0,Y 147.691,Z 699.113,A -85,B 0,C 180,E1 -23495.461,E2 -23495.461} C_VEL
LIN {X 0,Y 147.651,Z 699.875,A -85,B 0,C 180,E1 -23491.671,E2 -23491.671} C_VEL
LIN {X 0,Y 147.766,Z 699.973,A -85,B 0,C 180,E1 -23490,E2 -23490} C_VEL
LIN {X 0,Y 147.678,Z 699.755,A -85,B 0,C 180,E1 -23487.272,E2 -23487.272} C_VEL
LIN {X 0,Y 147.794,Z 699.14,A -85,B 0,C 180,E1 -23484.543,E2 -23484.543} C_VEL
LIN {X 0,Y 148.14,Z 698.134,A -85,B 0,C 180,E1 -23481.818,E2 -23481.818} C_VEL
LIN {X 0,Y 148.821,Z 696.717,A -85,B 0,C 180,E1 -23479.111,E2 -23479.111} C_VEL
LIN {X 0,Y 150.462,Z 693.762,A -85,B 0,C 180,E1 -23475.114,E2 -23475.114} C_VEL
LIN {X 0,Y 151.353,Z 692.607,A -85,B 0,C 180,E1 -23473.65,E2 -23473.65} C_VEL
